# B&R Automation Studio project reAM250plc (part 4)

#### TcpPacketHandler.hpp
```cpp
/*++

Copyright (C) 2024 Institute for Machine Tools and Industrial Management
TUM School of Engineering and Design
Technical University of Munich

All rights reserved.

Redistribution and use in source and binary forms, with or without
modification, are permitted provided that the following conditions are met:
	* Redistributions of source code must retain the above copyright
	  notice, this list of conditions and the following disclaimer.
	* Redistributions in binary form must reproduce the above copyright
	  notice, this list of conditions and the following disclaimer in the
	  documentation and/or other materials provided with the distribution.
	* Neither the name of the Technical University of Munich nor the
	  names of its contributors may be used to endorse or promote products
	  derived from this software without specific prior written permission.

THIS SOFTWARE IS PROVIDED BY THE COPYRIGHT HOLDERS AND CONTRIBUTORS "AS IS" AND
ANY EXPRESS OR IMPLIED WARRANTIES, INCLUDING, BUT NOT LIMITED TO, THE IMPLIED
WARRANTIES OF MERCHANTABILITY AND FITNESS FOR A PARTICULAR PURPOSE ARE
DISCLAIMED. IN NO EVENT SHALL TECHNICAL UNIVERSITY OF MUNICH BE LIABLE FOR ANY
DIRECT, INDIRECT, INCIDENTAL, SPECIAL, EXEMPLARY, OR CONSEQUENTIAL DAMAGES
(INCLUDING, BUT NOT LIMITED TO, PROCUREMENT OF SUBSTITUTE GOODS OR SERVICES;
LOSS OF USE, DATA, OR PROFITS; OR BUSINESS INTERRUPTION) HOWEVER CAUSED AND
ON ANY THEORY OF LIABILITY, WHETHER IN CONTRACT, STRICT LIABILITY, OR TORT
(INCLUDING NEGLIGENCE OR OTHERWISE) ARISING IN ANY WAY OUT OF THE USE OF THIS
SOFTWARE, EVEN IF ADVISED OF THE POSSIBILITY OF SUCH DAMAGE.

*/

#ifndef __TCPPACKETHANDLER_HPP
#define __TCPPACKETHANDLER_HPP

#include "Framework.hpp"
#include <list>
#include <vector>
#include <map>
#include <array>
#define	TCP_MAX_PACKET_RESPONSESIZE (256 * 1024)

namespace BuRCPP {

	class CTcpPacketResponse {
		private:
			std::array<uint8_t, TCP_MAX_PACKET_RESPONSESIZE> m_Payload;

			uint32_t m_nSignature;
			uint32_t m_nClientID;
			uint32_t m_nSequenceID;
			uint32_t m_nCurrentSize;
			uint32_t m_nErrorCode;

		public:

			CTcpPacketResponse ();
			virtual ~CTcpPacketResponse ();

			void addUint8 (uint8_t nValue);
			void addUint16 (uint16_t nValue);
			void addUint32 (uint32_t nValue);
			void addInt8 (int8_t nValue);
			void addInt16 (int16_t nValue);
			void addInt32 (int32_t nValue);
			void addDouble (double nValue);
			void addString (const std::string & sValue);
			void addPayload (uint8_t * pData, uint32_t nDataSize);

			void setErrorCode (eErrorCode nErrorCode);

			void beginResponse (uint32_t nClientID, uint32_t nSequenceID, uint32_t nSignature);
			void clearPayload ();

			uint32_t getClientID ();
			uint32_t getSequenceID ();
			uint32_t getCurrentSize ();

			std::array<uint8_t, TCP_MAX_PACKET_RESPONSESIZE> & getPayload ();

			void buildHeader (TcpOutgoingMessageHeader & header);

	};

	class CTcpPacketHandler {
		private:

		public:

		CTcpPacketHandler ();
		virtual ~CTcpPacketHandler();

		virtual uint32_t getCommandID () = 0;

		virtual bool isBufferedCommand () = 0;

		virtual void handlePacket (TcpIncomingPayload * pPayload, CTcpPacketResponse * pResponse) = 0;

		static uint8_t readUint8FromPayload (TcpIncomingPayload * pPayload, uint32_t nOffset);
		static uint16_t readUint16FromPayload (TcpIncomingPayload * pPayload, uint32_t nOffset);
		static uint32_t readUint32FromPayload (TcpIncomingPayload * pPayload, uint32_t nOffset);

	};

	class CTcpPacketHandler_Direct : public CTcpPacketHandler {
		public:

			CTcpPacketHandler_Direct ();

			virtual ~CTcpPacketHandler_Direct();

			virtual bool isBufferedCommand () override;

	};

	class CTcpPacketRegistry {
		private:

		std::map<uint32_t, std::shared_ptr<CTcpPacketHandler>> m_Handlers;
		uint32_t m_nPacketSignature;
		bool m_bPerformChecksumCheck;

		public:

		CTcpPacketRegistry (uint32_t nPacketSignature);

		virtual ~CTcpPacketRegistry();

		void registerHandler (std::shared_ptr<CTcpPacketHandler> pPacketHandler);

		bool canHandlePacket (uint32_t nCommandID);

		bool handlePacket (uint8_t * pData, uint32_t nDataSize, CTcpPacketResponse * pResponse);

	};

}

#endif // __TCPPACKETHANDLER_HPP
```

#### TcpPacketHandler.cpp
```cpp
/*++

Copyright (C) 2024 Institute for Machine Tools and Industrial Management
TUM School of Engineering and Design
Technical University of Munich

All rights reserved.

Redistribution and use in source and binary forms, with or without
modification, are permitted provided that the following conditions are met:
	* Redistributions of source code must retain the above copyright
	  notice, this list of conditions and the following disclaimer.
	* Redistributions in binary form must reproduce the above copyright
	  notice, this list of conditions and the following disclaimer in the
	  documentation and/or other materials provided with the distribution.
	* Neither the name of the Technical University of Munich nor the
	  names of its contributors may be used to endorse or promote products
	  derived from this software without specific prior written permission.

THIS SOFTWARE IS PROVIDED BY THE COPYRIGHT HOLDERS AND CONTRIBUTORS "AS IS" AND
ANY EXPRESS OR IMPLIED WARRANTIES, INCLUDING, BUT NOT LIMITED TO, THE IMPLIED
WARRANTIES OF MERCHANTABILITY AND FITNESS FOR A PARTICULAR PURPOSE ARE
DISCLAIMED. IN NO EVENT SHALL TECHNICAL UNIVERSITY OF MUNICH BE LIABLE FOR ANY
DIRECT, INDIRECT, INCIDENTAL, SPECIAL, EXEMPLARY, OR CONSEQUENTIAL DAMAGES
(INCLUDING, BUT NOT LIMITED TO, PROCUREMENT OF SUBSTITUTE GOODS OR SERVICES;
LOSS OF USE, DATA, OR PROFITS; OR BUSINESS INTERRUPTION) HOWEVER CAUSED AND
ON ANY THEORY OF LIABILITY, WHETHER IN CONTRACT, STRICT LIABILITY, OR TORT
(INCLUDING NEGLIGENCE OR OTHERWISE) ARISING IN ANY WAY OUT OF THE USE OF THIS
SOFTWARE, EVEN IF ADVISED OF THE POSSIBILITY OF SUCH DAMAGE.

*/

#include "TcpPacketHandler.hpp"
#include "Utils.hpp"

#include <bur/plctypes.h>

#ifdef _DEFAULT_INCLUDES
#include <AsDefault.h>
#endif

#include <string.h>

namespace BuRCPP
{

	CTcpPacketResponse::CTcpPacketResponse ()
	:  m_nSignature (0), m_nClientID (0), m_nSequenceID (0), m_nCurrentSize (0), m_nErrorCode (0)
	{
	}

	CTcpPacketResponse::~CTcpPacketResponse ()
	{
	}

	void CTcpPacketResponse::addPayload (uint8_t * pData, uint32_t nDataSize)
	{
		if ((pData != nullptr) && (nDataSize > 0)) {
			if (nDataSize > TCP_MAX_PACKET_RESPONSESIZE)
				throw CException (eErrorCode::INVALIDPARAM, "invalid packet response payload size.");

			uint32_t nNewDataSize = m_nCurrentSize + nDataSize;
			if (nNewDataSize > TCP_MAX_PACKET_RESPONSESIZE)
				throw CException (eErrorCode::INVALIDPARAM, "packet response payload overflow.");

			uint8_t * pSource = pData;
			uint8_t * pTarget = &m_Payload.at (m_nCurrentSize);

			for (uint32_t nIndex = 0; nIndex < nDataSize; nIndex++)
			{
				*pTarget = *pSource;
				pTarget++;
				pSource++;
			}

			m_nCurrentSize += nDataSize;

		}
	}

	void CTcpPacketResponse::addUint8 (uint8_t nValue)
	{
		addPayload ((uint8_t*)&nValue, sizeof (nValue));
	}

	void CTcpPacketResponse::addUint16 (uint16_t nValue)
	{
		addPayload ((uint8_t*)&nValue, sizeof (nValue));
	}

	void CTcpPacketResponse::addUint32 (uint32_t nValue)
	{
		addPayload ((uint8_t*)&nValue, sizeof (nValue));
	}

	void CTcpPacketResponse::addInt8 (int8_t nValue)
	{
		addPayload ((uint8_t*)&nValue, sizeof (nValue));
	}

	void CTcpPacketResponse::addInt16 (int16_t nValue)
	{
		addPayload ((uint8_t*)&nValue, sizeof (nValue));
	}

	void CTcpPacketResponse::addInt32 (int32_t nValue)
	{
		addPayload ((uint8_t*)&nValue, sizeof (nValue));
	}

	void CTcpPacketResponse::addDouble (double nValue)
	{
		addPayload ((uint8_t*)&nValue, sizeof (nValue));
	}

	void CTcpPacketResponse::addString (const std::string & sValue)
	{
		uint32_t nLength = sValue.length ();
		addPayload ((uint8_t*) sValue.c_str (), nLength);
	}

	void CTcpPacketResponse::setErrorCode (eErrorCode nErrorCode)
	{
		m_nErrorCode = (uint32_t) nErrorCode;
	}

	void CTcpPacketResponse::beginResponse (uint32_t nClientID, uint32_t nSequenceID, uint32_t nSignature)
	{
		m_nClientID = nClientID;
		m_nSequenceID = nSequenceID;
		m_nCurrentSize = 0;
		m_nSignature = nSignature;
		m_nErrorCode = 0;
	}

	uint32_t CTcpPacketResponse::getClientID ()
	{
		return m_nClientID;
	}

	uint32_t CTcpPacketResponse::getSequenceID ()
	{
		return m_nSequenceID;
	}

	uint32_t CTcpPacketResponse::getCurrentSize ()
	{
		return m_nCurrentSize;
	}

	std::array<uint8_t, TCP_MAX_PACKET_RESPONSESIZE> & CTcpPacketResponse::getPayload ()
	{
		return m_Payload;
	}

	void CTcpPacketResponse::buildHeader (TcpOutgoingMessageHeader & header)
	{

		header.m_nClientId = m_nClientID;
		header.m_nPayloadLength = (uint32_t) m_nCurrentSize;
		header.m_nSequenceId = m_nSequenceID;
		header.m_nSignature = m_nSignature;
		header.m_nStatusCode = m_nErrorCode;

		if (m_nCurrentSize > 0) {
			header.m_nPayloadChecksum = CUtils::computeCRC32 (m_Payload.data (), (uint32_t) m_nCurrentSize);
		} else {
			header.m_nPayloadChecksum = 0;
		}
		header.m_nHeaderChecksum = CUtils::computeCRC32 ((uint8_t*) &header, sizeof (header) - 4);
	}

	void CTcpPacketResponse::clearPayload ()
	{
		m_nCurrentSize = 0;
	}

	CTcpPacketHandler::CTcpPacketHandler ()
	{
	}

	CTcpPacketHandler::~CTcpPacketHandler()
	{
	}

	uint8_t CTcpPacketHandler::readUint8FromPayload (TcpIncomingPayload * pPayload, uint32_t nOffset)
	{
		if (pPayload == nullptr)
			throw CException (eErrorCode::INVALIDPARAM, "invalid packet payload param.");
		if (nOffset >= sizeof (TcpIncomingPayload))
			throw CException (eErrorCode::INVALIDPAYLOADOFFSET, "invalid packet payload offset.");

		return pPayload->m_Data[nOffset];
	}

	uint16_t CTcpPacketHandler::readUint16FromPayload (TcpIncomingPayload * pPayload, uint32_t nOffset)
	{
		if (pPayload == nullptr)
			throw CException (eErrorCode::INVALIDPARAM, "invalid packet payload param.");
		if ((nOffset + sizeof (uint16_t)) > sizeof (TcpIncomingPayload))
			throw CException (eErrorCode::INVALIDPAYLOADOFFSET, "invalid packet payload offset.");

		return *((uint16_t*)&pPayload->m_Data[nOffset]);
	}

	uint32_t CTcpPacketHandler::readUint32FromPayload (TcpIncomingPayload * pPayload, uint32_t nOffset)
	{
		if (pPayload == nullptr)
			throw CException (eErrorCode::INVALIDPARAM, "invalid packet payload param.");
		if ((nOffset + sizeof (uint32_t)) > sizeof (TcpIncomingPayload))
			throw CException (eErrorCode::INVALIDPAYLOADOFFSET, "invalid packet payload offset.");

		return *((uint32_t*)&pPayload->m_Data[nOffset]);

	}

	CTcpPacketHandler_Direct::CTcpPacketHandler_Direct ()
	: CTcpPacketHandler ()
	{
	}

	CTcpPacketHandler_Direct::~CTcpPacketHandler_Direct()
	{
	}

	bool CTcpPacketHandler_Direct::isBufferedCommand ()
	{
		return false;
	}

	CTcpPacketRegistry::CTcpPacketRegistry (uint32_t nPacketSignature)
		: m_nPacketSignature (nPacketSignature), m_bPerformChecksumCheck(false)
	{
	}

	CTcpPacketRegistry::~CTcpPacketRegistry()
	{
	}

	void CTcpPacketRegistry::registerHandler (std::shared_ptr<CTcpPacketHandler> pPacketHandler)
	{
		if (pPacketHandler.get () == nullptr)
			throw CException (eErrorCode::INVALIDPARAM, "invalid packet handler param.");

		uint32_t nCommand = pPacketHandler->getCommandID ();
		if (canHandlePacket (nCommand))
			throw CException (eErrorCode::PACKETHANDLERALREADYREGISTERED, "packet handler already registered: " + std::to_string (nCommand));

		m_Handlers.insert (std::make_pair (nCommand, pPacketHandler));

	}

	bool CTcpPacketRegistry::canHandlePacket (uint32_t nCommandID)
	{
		auto iIter = m_Handlers.find (nCommandID);
		return (iIter != m_Handlers.end ());
	}

	bool CTcpPacketRegistry::handlePacket (uint8_t * pData, uint32_t nDataSize, CTcpPacketResponse * pResponse)
	{

		if (pData == nullptr)
			throw CException (eErrorCode::INVALIDPARAM, "invalid packet data param.");
		if (nDataSize != sizeof (TcpIncomingMessage))
			throw CException (eErrorCode::INVALIDPARAM, "invalid packet data size param.");
		if (pResponse == nullptr)
			throw CException (eErrorCode::INVALIDPARAM, "invalid packet response pointer.");

		TcpIncomingMessage * pMessage = (TcpIncomingMessage*) pData;
		uint32_t nCommandID = pMessage->m_nCommandId;

		if(pMessage->m_nSignature != m_nPacketSignature)
			return false;

		if (m_bPerformChecksumCheck) {

			uint32_t nChecksum = CUtils::computeCRC32 ((uint8_t*)pMessage, (uint32_t)sizeof(TcpIncomingMessage) - 4);
			if(pMessage->m_nChecksum != nChecksum)
				return false;
		}

		auto iIter = m_Handlers.find (nCommandID);
		if (iIter == m_Handlers.end ())
			return false;

		CTcpPacketHandler * pHandler = iIter->second.get();
		pResponse->beginResponse (pMessage->m_nClientId, pMessage->m_nSequenceId, pMessage->m_nSignature);
		try {
			pHandler->handlePacket (&pMessage->m_Payload, pResponse);
			return true;

		}
		catch (CException & E) {
			pResponse->setErrorCode (E.getCode ());
			pResponse->clearPayload ();
		}

	}

}
```

#### TcpListHandler.hpp
```cpp
/*++

Copyright (C) 2024 Institute for Machine Tools and Industrial Management
TUM School of Engineering and Design
Technical University of Munich

All rights reserved.

Redistribution and use in source and binary forms, with or without
modification, are permitted provided that the following conditions are met:
	* Redistributions of source code must retain the above copyright
	  notice, this list of conditions and the following disclaimer.
	* Redistributions in binary form must reproduce the above copyright
	  notice, this list of conditions and the following disclaimer in the
	  documentation and/or other materials provided with the distribution.
	* Neither the name of the Technical University of Munich nor the
	  names of its contributors may be used to endorse or promote products
	  derived from this software without specific prior written permission.

THIS SOFTWARE IS PROVIDED BY THE COPYRIGHT HOLDERS AND CONTRIBUTORS "AS IS" AND
ANY EXPRESS OR IMPLIED WARRANTIES, INCLUDING, BUT NOT LIMITED TO, THE IMPLIED
WARRANTIES OF MERCHANTABILITY AND FITNESS FOR A PARTICULAR PURPOSE ARE
DISCLAIMED. IN NO EVENT SHALL TECHNICAL UNIVERSITY OF MUNICH BE LIABLE FOR ANY
DIRECT, INDIRECT, INCIDENTAL, SPECIAL, EXEMPLARY, OR CONSEQUENTIAL DAMAGES
(INCLUDING, BUT NOT LIMITED TO, PROCUREMENT OF SUBSTITUTE GOODS OR SERVICES;
LOSS OF USE, DATA, OR PROFITS; OR BUSINESS INTERRUPTION) HOWEVER CAUSED AND
ON ANY THEORY OF LIABILITY, WHETHER IN CONTRACT, STRICT LIABILITY, OR TORT
(INCLUDING NEGLIGENCE OR OTHERWISE) ARISING IN ANY WAY OUT OF THE USE OF THIS
SOFTWARE, EVEN IF ADVISED OF THE POSSIBILITY OF SUCH DAMAGE.

*/

#ifndef __TCPSYSTEMSTATE_HPP
#define __TCPSYSTEMSTATE_HPP

#include "Framework.hpp"
#include "TcpPacketHandler.hpp"
#include "SignalHandler.hpp"

#include <memory>

#define LISTCONTEXT_SIGNALSLOTCOUNT 16

namespace BuRCPP {

	enum class eListEntryState : int32_t {
		InQueue = 0,
		InitialExecution = 1,
		CyclicExecution = 2,
		Finished = 3,
		ExecutionError = 4
	};

	enum class eListState : int32_t {
		ListInQueue = 0,
		ListInCreation = 1,
		ListFinished = 2,
		ExecutingList = 3,
		ExecutionFinished = 4,
		ExecutionError = 5
	};

	typedef struct _TcpListEntryContext {
		eListEntryState m_nEntryState;
		uint32_t m_nLifeTimeInMilliseconds;
		CSignalSendInstance * m_pSignalSlots[LISTCONTEXT_SIGNALSLOTCOUNT];
		uint8_t m_ContextData[32];
	} TcpListEntryContext;

	class CTcpListHandler;

	class CSignalHandlerRegistry {
		private:
		public:

			virtual CSignalHandler * findSignalHandler (const std::string & sStateMachineName, bool bMustExist) = 0;
	};

	class CPayloadEnvironment
	{
		private:

		TcpListEntryContext * m_pContext;
		TcpIncomingPayload * m_pPayload;
		CSignalHandlerRegistry * m_pSignalHandlerRegistry;

		public:

		CPayloadEnvironment (TcpListEntryContext * pContext, TcpIncomingPayload * pPayload, CSignalHandlerRegistry * pSignalHandlerRegistry);

		virtual ~CPayloadEnvironment ();

		eListEntryState getState ();

		bool isFirstCycle ();

		uint32_t getPayloadSize ();

		void readPayloadData (uint8_t * pTarget, uint32_t nAddress, uint32_t nByteCount);
		uint8_t readPayloadUint8 (uint32_t nAddress);
		uint16_t readPayloadUint16 (uint32_t nAddress);
		uint32_t readPayloadUint32 (uint32_t nAddress);
		int8_t readPayloadInt8 (uint32_t nAddress);
		int16_t readPayloadInt16 (uint32_t nAddress);
		int32_t readPayloadInt32 (uint32_t nAddress);
		double readPayloadDouble (uint32_t nAddress);
		float readPayloadFloat (uint32_t nAddress);

		uint32_t getContextSize ();

		void readContextData (uint8_t * pTarget, uint32_t nAddress, uint32_t nByteCount);
		uint8_t readContextUint8 (uint32_t nAddress);
		uint16_t readContextUint16 (uint32_t nAddress);
		uint32_t readContextUint32 (uint32_t nAddress);
		int8_t readContextInt8 (uint32_t nAddress);
		int16_t readContextInt16 (uint32_t nAddress);
		int32_t readContextInt32 (uint32_t nAddress);
		double readContextDouble (uint32_t nAddress);
		float readContextFloat (uint32_t nAddress);

		void writeContextData (uint8_t * pSource, uint32_t nAddress, uint32_t nByteCount);
		void writeContextUint8 (uint32_t nAddress, uint8_t nValue);
		void writeContextUint16 (uint32_t nAddress, uint16_t nValue);
		void writeContextUint32 (uint32_t nAddress, uint32_t nValue);
		void writeContextInt8 (uint32_t nAddress, int8_t nValue);
		void writeContextInt16 (uint32_t nAddress, int16_t nValue);
		void writeContextInt32 (uint32_t nAddress, int32_t nValue);
		void writeContextDouble (uint32_t nAddress, double dValue);
		void writeContextFloat (uint32_t nAddress, float dValue);

		void setLifetimeInMillseconds (uint32_t nLifeTimeInMilliseconds);

		CSignalSendInstance * prepareSignal (uint32_t nSignalSlotIndex, const std::string & sStateHandlerName, const std::string & sSignalName);
		CSignalSendInstance * getSignal (uint32_t nSignalSlotIndex, bool bMustExist);
		bool signalHasBeenProcessed (uint32_t nSignalSlotIndex);

	};

	class CTcpPacketHandler_Buffered : public CTcpPacketHandler {

		private:
		CTcpListHandler * m_pListHandler;

		public:

		CTcpPacketHandler_Buffered (CTcpListHandler * pListHandler);

		virtual ~CTcpPacketHandler_Buffered();

		virtual bool isBufferedCommand () override;

		virtual void handlePacket (TcpIncomingPayload * pPayload, CTcpPacketResponse * pResponse) override;

		virtual void enterExecution (CPayloadEnvironment * pEnvironment);

		virtual bool cyclicExecution (CPayloadEnvironment * pEnvironment);

	};

	struct _TcpListEntry;
	typedef struct _TcpListEntry TcpListEntry;

	struct _TcpList;
	typedef struct _TcpList TcpList;

	struct _TcpListEntry {
		CTcpPacketHandler_Buffered * m_PacketHandler;
		TcpIncomingPayload m_Payload;
		uint32_t m_nIndexInList;
		TcpListEntryContext m_ExecutionContext;
		TcpListEntry * m_pNext;
	};

	struct _TcpList {
		uint32_t m_nListId;
		uint32_t m_nEntryCount;
		eListState m_ListState;
		TcpListEntry * m_pFirstEntry;
		TcpListEntry * m_pLastEntry;
		TcpListEntry * m_pCurrentEntry;
		TcpList * m_pNextUnusedList;
	};

	class CTcpListHandler {

		private:
		std::vector<TcpListEntry> m_ListEntryBuffer;
		std::vector<TcpList> m_ListBuffer;
		TcpList * m_pUnusedLists;
		TcpListEntry * m_pUnusedListEntries;

		TcpList * m_pCurrentWriteList;

		TcpList * m_pCurrentExecutionList;

		CSignalHandlerRegistry * m_pSignalHandlerRegistry;

		void addEntryToList (TcpList *, CTcpPacketHandler_Buffered * pHandler, TcpIncomingPayload * pPayload);

		public:

		CTcpListHandler (uint32_t nListBufferSize, uint32_t nListEntryBufferSize, CSignalHandlerRegistry * pSignalHandlerRegistry);

		virtual ~CTcpListHandler ();

		void registerDefaultCommands (CTcpPacketRegistry * pPacketRegistry);

		uint32_t beginList ();
		TcpList * finishList ();
		TcpList* executeList (uint32_t nListID);
		TcpList* getListByID (uint32_t nListID, bool bListMustExist);

		bool hasCurrentList ();

		TcpListEntry * addCommandToCurrentList (CTcpPacketHandler_Buffered * pHandler, TcpIncomingPayload * pPayload);

		void handleCyclic ();

	};

}

#endif // __TCPSYSTEMSTATE_HPP
```

#### TcpListHandler.cpp
```cpp
/*++

Copyright (C) 2024 Institute for Machine Tools and Industrial Management
TUM School of Engineering and Design
Technical University of Munich

All rights reserved.

Redistribution and use in source and binary forms, with or without
modification, are permitted provided that the following conditions are met:
	* Redistributions of source code must retain the above copyright
	  notice, this list of conditions and the following disclaimer.
	* Redistributions in binary form must reproduce the above copyright
	  notice, this list of conditions and the following disclaimer in the
	  documentation and/or other materials provided with the distribution.
	* Neither the name of the Technical University of Munich nor the
	  names of its contributors may be used to endorse or promote products
	  derived from this software without specific prior written permission.

THIS SOFTWARE IS PROVIDED BY THE COPYRIGHT HOLDERS AND CONTRIBUTORS "AS IS" AND
ANY EXPRESS OR IMPLIED WARRANTIES, INCLUDING, BUT NOT LIMITED TO, THE IMPLIED
WARRANTIES OF MERCHANTABILITY AND FITNESS FOR A PARTICULAR PURPOSE ARE
DISCLAIMED. IN NO EVENT SHALL TECHNICAL UNIVERSITY OF MUNICH BE LIABLE FOR ANY
DIRECT, INDIRECT, INCIDENTAL, SPECIAL, EXEMPLARY, OR CONSEQUENTIAL DAMAGES
(INCLUDING, BUT NOT LIMITED TO, PROCUREMENT OF SUBSTITUTE GOODS OR SERVICES;
LOSS OF USE, DATA, OR PROFITS; OR BUSINESS INTERRUPTION) HOWEVER CAUSED AND
ON ANY THEORY OF LIABILITY, WHETHER IN CONTRACT, STRICT LIABILITY, OR TORT
(INCLUDING NEGLIGENCE OR OTHERWISE) ARISING IN ANY WAY OUT OF THE USE OF THIS
SOFTWARE, EVEN IF ADVISED OF THE POSSIBILITY OF SUCH DAMAGE.

*/

#include "TcpListHandler.hpp"

#include <cstring>

namespace BuRCPP {

	CPayloadEnvironment::CPayloadEnvironment (TcpListEntryContext * pContext, TcpIncomingPayload * pPayload, CSignalHandlerRegistry * pSignalHandlerRegistry)
		: m_pContext (pContext), m_pPayload (pPayload), m_pSignalHandlerRegistry (pSignalHandlerRegistry)
	{
		if ((pContext == nullptr) || (pPayload == nullptr) || (pSignalHandlerRegistry == nullptr))
			throw CException (eErrorCode::INVALIDPARAM, "invalid payload environment parameters");

	}

	CPayloadEnvironment::~CPayloadEnvironment ()
	{
	}

	eListEntryState CPayloadEnvironment::getState ()
	{
		return m_pContext->m_nEntryState;
	}

	bool CPayloadEnvironment::isFirstCycle ()
	{
		return m_pContext->m_nEntryState == eListEntryState::InitialExecution;
	}

	uint32_t CPayloadEnvironment::getPayloadSize ()
	{
		return sizeof (TcpIncomingPayload);
	}

	void CPayloadEnvironment::readPayloadData (uint8_t * pTarget, uint32_t nAddress, uint32_t nByteCount)
	{
		if (nByteCount == 0)
			return;

		if (pTarget == nullptr)
			throw CException (eErrorCode::INVALIDPARAM, "invalid read payload target parameter");

		if (nAddress >=  sizeof (TcpIncomingPayload))
			throw CException (eErrorCode::INVALIDPAYLOADADDRESS, "invalid payload address");

		if (nByteCount >=  sizeof (TcpIncomingPayload))
			throw CException (eErrorCode::INVALIDPAYLOADREADOPERATION, "invalid payload read size");
		if ((nAddress + nByteCount) > sizeof (TcpIncomingPayload))
			throw CException (eErrorCode::INVALIDPAYLOADREADOPERATION, "payload read buffer overflow");

		for (uint32_t nIndex = 0; nIndex < nByteCount; nIndex++)
			pTarget[nIndex] = m_pPayload->m_Data[nAddress + nIndex];

	}

	uint8_t CPayloadEnvironment::readPayloadUint8 (uint32_t nAddress)
	{
		uint8_t nResult = 0;
		readPayloadData ((uint8_t*)&nResult, nAddress, sizeof (nResult));
		return nResult;
	}

	uint16_t CPayloadEnvironment::readPayloadUint16 (uint32_t nAddress)
	{
		uint16_t nResult = 0;
		readPayloadData ((uint8_t*)&nResult, nAddress, sizeof (nResult));
		return nResult;
	}

	uint32_t CPayloadEnvironment::readPayloadUint32 (uint32_t nAddress)
	{
		uint32_t nResult = 0;
		readPayloadData ((uint8_t*)&nResult, nAddress, sizeof (nResult));
		return nResult;
	}

	int8_t CPayloadEnvironment::readPayloadInt8 (uint32_t nAddress)
	{
		int8_t nResult = 0;
		readPayloadData ((uint8_t*)&nResult, nAddress, sizeof (nResult));
		return nResult;
	}

	int16_t CPayloadEnvironment::readPayloadInt16 (uint32_t nAddress)
	{
		int16_t nResult = 0;
		readPayloadData ((uint8_t*)&nResult, nAddress, sizeof (nResult));
		return nResult;
	}

	int32_t CPayloadEnvironment::readPayloadInt32 (uint32_t nAddress)
	{
		uint32_t nResult = 0;
		readPayloadData ((uint8_t*)&nResult, nAddress, sizeof (nResult));
		return nResult;

	}

	double CPayloadEnvironment::readPayloadDouble (uint32_t nAddress)
	{
		double dResult = 0.0;
		readPayloadData ((uint8_t*)&dResult, nAddress, sizeof (dResult));
		return dResult;

	}

	float CPayloadEnvironment::readPayloadFloat (uint32_t nAddress)
	{
		float fResult = 0.0;
		readPayloadData ((uint8_t*)&fResult, nAddress, sizeof (fResult));
		return fResult;

	}

	uint32_t CPayloadEnvironment::getContextSize ()
	{
		return sizeof (m_pContext->m_ContextData);
	}

	void CPayloadEnvironment::readContextData (uint8_t * pTarget, uint32_t nAddress, uint32_t nByteCount)
	{
	}

	uint8_t CPayloadEnvironment::readContextUint8 (uint32_t nAddress)
	{

	}

	uint16_t CPayloadEnvironment::readContextUint16 (uint32_t nAddress)
	{

	}

	uint32_t CPayloadEnvironment::readContextUint32 (uint32_t nAddress)
	{

	}

	int8_t CPayloadEnvironment::readContextInt8 (uint32_t nAddress)
	{

	}

	int16_t CPayloadEnvironment::readContextInt16 (uint32_t nAddress)
	{

	}

	int32_t CPayloadEnvironment::readContextInt32 (uint32_t nAddress)
	{

	}

	double CPayloadEnvironment::readContextDouble (uint32_t nAddress)
	{

	}

	float CPayloadEnvironment::readContextFloat (uint32_t nAddress)
	{

	}

	void CPayloadEnvironment::writeContextData (uint8_t * pSource, uint32_t nAddress, uint32_t nByteCount)
	{

	}

	void CPayloadEnvironment::writeContextUint8 (uint32_t nAddress, uint8_t nValue)
	{
	}

	void CPayloadEnvironment::writeContextUint16 (uint32_t nAddress, uint16_t nValue)
	{
	}

	void CPayloadEnvironment::writeContextUint32 (uint32_t nAddress, uint32_t nValue)
	{
	}

	void CPayloadEnvironment::writeContextInt8 (uint32_t nAddress, int8_t nValue)
	{
	}

	void CPayloadEnvironment::writeContextInt16 (uint32_t nAddress, int16_t nValue)
	{
	}

	void CPayloadEnvironment::writeContextInt32 (uint32_t nAddress, int32_t nValue)
	{
	}

	void CPayloadEnvironment::writeContextDouble (uint32_t nAddress, double dValue)
	{
	}

	void CPayloadEnvironment::writeContextFloat (uint32_t nAddress, float dValue)
	{
	}

	void CPayloadEnvironment::setLifetimeInMillseconds (uint32_t nLifeTimeInMilliseconds)
	{
		m_pContext->m_nLifeTimeInMilliseconds = nLifeTimeInMilliseconds;
	}

	CSignalSendInstance * CPayloadEnvironment::prepareSignal (uint32_t nSignalSlotIndex, const std::string & sStateHandlerName, const std::string & sSignalName)
	{
		if (nSignalSlotIndex >= LISTCONTEXT_SIGNALSLOTCOUNT)
			throw CException (eErrorCode::INVALIDSIGNALSLOTINDEX, "invalid payload signal slot index: " + std::to_string (nSignalSlotIndex));

		if (m_pContext->m_pSignalSlots[nSignalSlotIndex] != nullptr)
			throw CException (eErrorCode::PAYLOADSIGNALSLOTALREADYTAKEN, "signal slot already taken: " + std::to_string (nSignalSlotIndex));

		auto pSignalHandler = m_pSignalHandlerRegistry->findSignalHandler (sStateHandlerName, true);

		CSignalSendInstance * pSignalInstance = pSignalHandler->prepareSignal (sSignalName);

		m_pContext->m_pSignalSlots[nSignalSlotIndex] = pSignalInstance;

		return pSignalInstance;
	}

	CSignalSendInstance * CPayloadEnvironment::getSignal (uint32_t nSignalSlotIndex, bool bMustExist)
	{
		if (nSignalSlotIndex >= LISTCONTEXT_SIGNALSLOTCOUNT)
			throw CException (eErrorCode::INVALIDSIGNALSLOTINDEX, "invalid payload signal slot index: " + std::to_string (nSignalSlotIndex));

		CSignalSendInstance * pSignalInstance =	m_pContext->m_pSignalSlots[nSignalSlotIndex];
		if ((pSignalInstance == nullptr) && bMustExist)
			throw CException (eErrorCode::SIGNALSLOTISEMPTY, "payload signal slot is empty: " + std::to_string (nSignalSlotIndex));

		return pSignalInstance;
	}

	bool CPayloadEnvironment::signalHasBeenProcessed (uint32_t nSignalSlot)
	{
		CSignalSendInstance * pSignalInstance = getSignal (nSignalSlot, true);
		return pSignalInstance->signalHasBeenProcessed ();
	}

	class CTcpPacketHandler_BeginList : public CTcpPacketHandler_Direct {
		private:
			CTcpListHandler* m_pListHandler;

		public:

			CTcpPacketHandler_BeginList (CTcpListHandler * pListHandler)
			: CTcpPacketHandler_Direct (), m_pListHandler (pListHandler)
				{
				}

			virtual ~CTcpPacketHandler_BeginList ()
			{
			}

			virtual uint32_t getCommandID () override
			{
				return COMMAND_DEFAULT_BEGINLIST;
			}

			void handlePacket (TcpIncomingPayload * pPayload, CTcpPacketResponse * pResponse) override
			{
				beginListCalled++;
				pResponse->addUint32(m_pListHandler->beginList ());
			}

	};

	class CTcpPacketHandler_FinishList : public CTcpPacketHandler_Direct {
		private:
		CTcpListHandler* m_pListHandler;

		public:

		CTcpPacketHandler_FinishList (CTcpListHandler * pListHandler)
			: CTcpPacketHandler_Direct (), m_pListHandler (pListHandler)
		{
		}

		virtual ~CTcpPacketHandler_FinishList ()
		{
		}

		virtual uint32_t getCommandID () override
		{
			return COMMAND_DEFAULT_FINISHLIST;
		}

			void handlePacket (TcpIncomingPayload * pPayload, CTcpPacketResponse * pResponse) override
			{
				finishListCalled++;
				TcpList* pList = m_pListHandler->finishList ();
				pResponse->addUint32(pList->m_nListId);
				pResponse->addUint32(pList->m_nEntryCount);
			}

	};

	class CTcpPacketHandler_ExecuteList : public CTcpPacketHandler_Direct {
		private:
		CTcpListHandler* m_pListHandler;

		public:

		CTcpPacketHandler_ExecuteList (CTcpListHandler * pListHandler)
			: CTcpPacketHandler_Direct (), m_pListHandler (pListHandler)
		{
		}

		virtual ~CTcpPacketHandler_ExecuteList ()
		{
		}

		virtual uint32_t getCommandID () override
		{
			return COMMAND_DEFAULT_EXECUTELIST;
		}

		void handlePacket (TcpIncomingPayload * pPayload, CTcpPacketResponse * pResponse) override
		{
			uint32_t nListID = readUint32FromPayload (pPayload, 0);
			TcpList * pList = m_pListHandler->executeList (nListID);

			pResponse->addUint32(pList->m_nEntryCount);
		}
	};

		class CTcpPacketHandler_ListStatus : public CTcpPacketHandler_Direct {
			private:
			CTcpListHandler* m_pListHandler;

			public:

				CTcpPacketHandler_ListStatus (CTcpListHandler * pListHandler)
					: CTcpPacketHandler_Direct (), m_pListHandler (pListHandler)
				{
				}

				virtual ~CTcpPacketHandler_ListStatus ()
				{
				}

				virtual uint32_t getCommandID () override
				{
					return COMMAND_DEFAULT_LISTSTATUS;
				}

				void handlePacket (TcpIncomingPayload * pPayload, CTcpPacketResponse * pResponse) override
				{
					uint32_t nListID = readUint32FromPayload (pPayload, 0);
					TcpList * pList = m_pListHandler->getListByID (nListID, false);

					if (pList != nullptr) {
						pResponse->addUint32(pList->m_nListId);
						pResponse->addUint32((uint32_t)pList->m_ListState);
						pResponse->addUint32(pList->m_nEntryCount);
						if (pList->m_pCurrentEntry != nullptr) {
							pResponse->addUint32(pList->m_pCurrentEntry->m_nIndexInList);
						} else {
							pResponse->addUint32(0);
						}

					} else {
						pResponse->addUint32(0);
						pResponse->addUint32(0);
						pResponse->addUint32(0);
						pResponse->addUint32(0);
					}

				}

	};

CTcpPacketHandler_Buffered::CTcpPacketHandler_Buffered (CTcpListHandler * pListHandler)
	: CTcpPacketHandler (), m_pListHandler (pListHandler)
{
}

CTcpPacketHandler_Buffered::~CTcpPacketHandler_Buffered()
{
}

bool CTcpPacketHandler_Buffered::isBufferedCommand ()
{
	return true;
}

void CTcpPacketHandler_Buffered::handlePacket (TcpIncomingPayload * pPayload, CTcpPacketResponse * pResponse)
{
	TcpListEntry* pNewEntry = m_pListHandler->addCommandToCurrentList (this, pPayload);
	pResponse->addUint32(pNewEntry->m_nIndexInList);

}

void CTcpPacketHandler_Buffered::enterExecution (CPayloadEnvironment * pEnvironment)
{

}

bool CTcpPacketHandler_Buffered::cyclicExecution (CPayloadEnvironment * pEnvironment)
{
	return true;
}

	CTcpListHandler::CTcpListHandler (uint32_t nListBufferSize, uint32_t nListEntryBufferSize, CSignalHandlerRegistry * pSignalHandlerRegistry)
	: m_pUnusedLists (nullptr), m_pUnusedListEntries (nullptr), m_pCurrentWriteList (nullptr), m_pCurrentExecutionList (nullptr), m_pSignalHandlerRegistry (pSignalHandlerRegistry)
	{

		if (pSignalHandlerRegistry == nullptr)
			throw std::runtime_error ("invalid signal handler registry param");

		m_ListEntryBuffer.resize (nListEntryBufferSize);
		m_ListBuffer.resize (nListBufferSize);

		uint32_t nListIndex = nListBufferSize;
		while (nListIndex > 0) {
			nListIndex--;

			auto pList = &m_ListBuffer[nListIndex];
			pList->m_nListId = nListIndex + 1;
			pList->m_nEntryCount = 0;
			pList->m_pLastEntry = nullptr;
			pList->m_pFirstEntry = nullptr;
			pList->m_pCurrentEntry = nullptr;
			pList->m_ListState = eListState::ListInQueue;

			pList->m_pNextUnusedList = m_pUnusedLists;
			m_pUnusedLists = pList;

		}

		uint32_t nListEntryIndex = nListEntryBufferSize;
		while (nListEntryIndex > 0) {
			nListEntryIndex--;

			auto pListEntry = &m_ListEntryBuffer[nListEntryIndex];
			pListEntry->m_pNext = m_pUnusedListEntries;
			pListEntry->m_PacketHandler = nullptr;
			pListEntry->m_nIndexInList = 0;
			memset ((void*) &pListEntry->m_Payload, 0, sizeof (pListEntry->m_Payload));
			m_pUnusedListEntries = pListEntry;

		}
	}

	CTcpListHandler::~CTcpListHandler ()
	{
	}

	void CTcpListHandler::registerDefaultCommands (CTcpPacketRegistry * pPacketRegistry)
	{
		if (pPacketRegistry == nullptr)
			throw CException (eErrorCode::INVALIDPARAM, "invalid packet registry parameter");

		pPacketRegistry->registerHandler (std::make_shared<CTcpPacketHandler_BeginList> (this));
		pPacketRegistry->registerHandler (std::make_shared<CTcpPacketHandler_FinishList> (this));
		pPacketRegistry->registerHandler (std::make_shared<CTcpPacketHandler_ExecuteList> (this));
		pPacketRegistry->registerHandler (std::make_shared<CTcpPacketHandler_ListStatus> (this));

	}

	uint32_t CTcpListHandler::beginList ()
	{
		if (m_pUnusedLists == nullptr)
			throw CException (eErrorCode::TOOMANYOPENLISTS, "too many open lists!");

		if (m_pUnusedLists->m_ListState != eListState::ListInQueue)
			throw CException (eErrorCode::LISTISNOTINQUEUE, "list is not in queue!");

		m_pCurrentWriteList = m_pUnusedLists;
		m_pUnusedLists = m_pUnusedLists->m_pNextUnusedList;

		m_pCurrentWriteList->m_nEntryCount = 0;
		m_pCurrentWriteList->m_pCurrentEntry = nullptr;
		m_pCurrentWriteList->m_pFirstEntry = nullptr;
		m_pCurrentWriteList->m_pLastEntry = nullptr;
		m_pCurrentWriteList->m_pNextUnusedList = nullptr;
		m_pCurrentWriteList->m_ListState = eListState::ListInCreation;

		return m_pCurrentWriteList->m_nListId;
	}

	TcpList* CTcpListHandler::finishList ()
	{

		if (m_pCurrentWriteList == nullptr)
			throw CException (eErrorCode::NOTWRITINGTOANYLIST, "not writing to any list!");
		if (m_pCurrentWriteList->m_ListState != eListState::ListInCreation)
			throw CException (eErrorCode::NOTINLISTCREATION, "list not in creation!");
		if (m_pCurrentWriteList->m_pFirstEntry == nullptr)
			throw CException (eErrorCode::LISTISEMPTY, "list is empty!");

		auto pList = m_pCurrentWriteList;
		m_pCurrentWriteList = nullptr;

		pList->m_ListState = eListState::ListFinished;
		return pList;
	}

	TcpList* CTcpListHandler::getListByID (uint32_t nListID, bool bListMustExist)
	{
		TcpList * pList = nullptr;
		if ((nListID > 0) || (nListID <= m_ListBuffer.size ())) {
			pList = &m_ListBuffer.at (nListID - 1);
			if (pList->m_ListState == eListState::ListInQueue)
				pList = nullptr;
		}

		if ((pList == nullptr) && bListMustExist)
			throw CException (eErrorCode::LISTDOESNOTEXIST, "list does not exist");

		return pList;
	}

	TcpList* CTcpListHandler::executeList (uint32_t nListID)
	{
		m_pCurrentExecutionList = nullptr;

		if ((nListID == 0) || (nListID > m_ListBuffer.size ()))
			throw CException (eErrorCode::INVALIDLISTID, "invalid list ID");

		auto pList = &m_ListBuffer.at (nListID - 1);
		if (pList->m_ListState != eListState::ListFinished)
			throw CException (eErrorCode::LISTISNOTFINISHED, "list is not in finished!");
		if (pList->m_pFirstEntry == nullptr)
			throw CException (eErrorCode::LISTISEMPTY, "list is empty!");

		m_pCurrentExecutionList = pList;
		m_pCurrentExecutionList->m_pCurrentEntry = m_pCurrentExecutionList->m_pFirstEntry;
		m_pCurrentExecutionList->m_ListState = eListState::ExecutingList;

		return m_pCurrentExecutionList;
	}

	bool CTcpListHandler::hasCurrentList ()
	{
		return (m_pCurrentWriteList != nullptr);
	}

	TcpListEntry* CTcpListHandler::addCommandToCurrentList (CTcpPacketHandler_Buffered * pHandler, TcpIncomingPayload * pPayload)
	{
		if (pHandler == nullptr)
			throw CException (eErrorCode::INVALIDPARAM, "invalid packet handler parameter");
		if (pPayload == nullptr)
			throw CException (eErrorCode::INVALIDPAYLOAD, "invalid payload.");
		if (m_pCurrentWriteList == nullptr)
			throw CException (eErrorCode::NOLISTTOWRITETO, "no list to write to.");
		if (m_pUnusedListEntries == nullptr)
			throw CException (eErrorCode::NOLISTENTRIESLEFT, "no list entries left");

		auto pNewListEntry = m_pUnusedListEntries;
		m_pUnusedListEntries = m_pUnusedListEntries->m_pNext;

		pNewListEntry->m_PacketHandler = pHandler;
		pNewListEntry->m_Payload = *pPayload;
		pNewListEntry->m_pNext = nullptr;
		pNewListEntry->m_nIndexInList = m_pCurrentWriteList->m_nEntryCount;

		memset ((void*)&pNewListEntry->m_ExecutionContext, 0, sizeof (pNewListEntry->m_ExecutionContext));
		pNewListEntry->m_ExecutionContext.m_nEntryState = eListEntryState::InQueue;

		m_pCurrentWriteList->m_nEntryCount++;
		if (m_pCurrentWriteList->m_pFirstEntry == nullptr)
			m_pCurrentWriteList->m_pFirstEntry = pNewListEntry;
		if (m_pCurrentWriteList->m_pLastEntry != nullptr)
			m_pCurrentWriteList->m_pLastEntry->m_pNext = pNewListEntry;
		m_pCurrentWriteList->m_pLastEntry = pNewListEntry;

		bufferedListEntries++;

		return pNewListEntry;
	}

	void CTcpListHandler::handleCyclic ()
	{
		if (m_pCurrentExecutionList != nullptr) {

			auto pEntryToExecute = m_pCurrentExecutionList->m_pCurrentEntry;
			if (pEntryToExecute != nullptr) {
				switch (pEntryToExecute->m_ExecutionContext.m_nEntryState) {
					case eListEntryState::InQueue:
					{
						pEntryToExecute->m_ExecutionContext.m_nEntryState = eListEntryState::InitialExecution;
						break;
					}

					case eListEntryState::InitialExecution:
					{
						try {

							if (pEntryToExecute->m_PacketHandler == nullptr)
								throw CException (eErrorCode::INTERNALLISTERROR, "internal list error");

							CPayloadEnvironment environment (&pEntryToExecute->m_ExecutionContext, &pEntryToExecute->m_Payload, m_pSignalHandlerRegistry);

							pEntryToExecute->m_PacketHandler->enterExecution (&environment);
							pEntryToExecute->m_ExecutionContext.m_nEntryState = eListEntryState::CyclicExecution;

						} catch (...) {
							pEntryToExecute->m_ExecutionContext.m_nEntryState = eListEntryState::ExecutionError;
						}

						break;
					}

					case eListEntryState::CyclicExecution:
					{
						try {

							if (pEntryToExecute->m_PacketHandler == nullptr)
								throw CException (eErrorCode::INTERNALLISTERROR, "internal list error");

							CPayloadEnvironment environment (&pEntryToExecute->m_ExecutionContext, &pEntryToExecute->m_Payload, m_pSignalHandlerRegistry);

							bool bIsFinished = pEntryToExecute->m_PacketHandler->cyclicExecution (&environment);
							if (bIsFinished) {
								pEntryToExecute->m_ExecutionContext.m_nEntryState = eListEntryState::Finished;
							} else {
								pEntryToExecute->m_ExecutionContext.m_nEntryState = eListEntryState::CyclicExecution;
							}

						} catch (...) {
							pEntryToExecute->m_ExecutionContext.m_nEntryState = eListEntryState::ExecutionError;
						}

						break;
					}

					case eListEntryState::Finished:
					{
						m_pCurrentExecutionList->m_pCurrentEntry = pEntryToExecute->m_pNext;
						break;
					}

					case eListEntryState::ExecutionError:
					{
						m_pCurrentExecutionList = nullptr;
						break;
					}

				}

			}

		}
	}

}
```

#### Utils.hpp
```cpp
/*++

Copyright (C) 2024 Institute for Machine Tools and Industrial Management
TUM School of Engineering and Design
Technical University of Munich

All rights reserved.

Redistribution and use in source and binary forms, with or without
modification, are permitted provided that the following conditions are met:
	* Redistributions of source code must retain the above copyright
	  notice, this list of conditions and the following disclaimer.
	* Redistributions in binary form must reproduce the above copyright
	  notice, this list of conditions and the following disclaimer in the
	  documentation and/or other materials provided with the distribution.
	* Neither the name of the Technical University of Munich nor the
	  names of its contributors may be used to endorse or promote products
	  derived from this software without specific prior written permission.

THIS SOFTWARE IS PROVIDED BY THE COPYRIGHT HOLDERS AND CONTRIBUTORS "AS IS" AND
ANY EXPRESS OR IMPLIED WARRANTIES, INCLUDING, BUT NOT LIMITED TO, THE IMPLIED
WARRANTIES OF MERCHANTABILITY AND FITNESS FOR A PARTICULAR PURPOSE ARE
DISCLAIMED. IN NO EVENT SHALL TECHNICAL UNIVERSITY OF MUNICH BE LIABLE FOR ANY
DIRECT, INDIRECT, INCIDENTAL, SPECIAL, EXEMPLARY, OR CONSEQUENTIAL DAMAGES
(INCLUDING, BUT NOT LIMITED TO, PROCUREMENT OF SUBSTITUTE GOODS OR SERVICES;
LOSS OF USE, DATA, OR PROFITS; OR BUSINESS INTERRUPTION) HOWEVER CAUSED AND
ON ANY THEORY OF LIABILITY, WHETHER IN CONTRACT, STRICT LIABILITY, OR TORT
(INCLUDING NEGLIGENCE OR OTHERWISE) ARISING IN ANY WAY OUT OF THE USE OF THIS
SOFTWARE, EVEN IF ADVISED OF THE POSSIBILITY OF SUCH DAMAGE.

*/

#ifndef __UTILS_HPP
#define __UTILS_HPP

#include "Framework.hpp"
#include <memory>

namespace BuRCPP {

	class CUtils {

	public:

		static uint32_t computeCRC32 (uint8_t * pBuf, uint32_t len);

		static void writeStringVariable(const std::string & sString, char * pVariable, uint32_t nCount);

	};

}

#endif // __UTILS_HPP
```

#### Utils.cpp
```cpp
/*++

Copyright (C) 2024 Institute for Machine Tools and Industrial Management
TUM School of Engineering and Design
Technical University of Munich

All rights reserved.

Redistribution and use in source and binary forms, with or without
modification, are permitted provided that the following conditions are met:
	* Redistributions of source code must retain the above copyright
	  notice, this list of conditions and the following disclaimer.
	* Redistributions in binary form must reproduce the above copyright
	  notice, this list of conditions and the following disclaimer in the
	  documentation and/or other materials provided with the distribution.
	* Neither the name of the Technical University of Munich nor the
	  names of its contributors may be used to endorse or promote products
	  derived from this software without specific prior written permission.

THIS SOFTWARE IS PROVIDED BY THE COPYRIGHT HOLDERS AND CONTRIBUTORS "AS IS" AND
ANY EXPRESS OR IMPLIED WARRANTIES, INCLUDING, BUT NOT LIMITED TO, THE IMPLIED
WARRANTIES OF MERCHANTABILITY AND FITNESS FOR A PARTICULAR PURPOSE ARE
DISCLAIMED. IN NO EVENT SHALL TECHNICAL UNIVERSITY OF MUNICH BE LIABLE FOR ANY
DIRECT, INDIRECT, INCIDENTAL, SPECIAL, EXEMPLARY, OR CONSEQUENTIAL DAMAGES
(INCLUDING, BUT NOT LIMITED TO, PROCUREMENT OF SUBSTITUTE GOODS OR SERVICES;
LOSS OF USE, DATA, OR PROFITS; OR BUSINESS INTERRUPTION) HOWEVER CAUSED AND
ON ANY THEORY OF LIABILITY, WHETHER IN CONTRACT, STRICT LIABILITY, OR TORT
(INCLUDING NEGLIGENCE OR OTHERWISE) ARISING IN ANY WAY OUT OF THE USE OF THIS
SOFTWARE, EVEN IF ADVISED OF THE POSSIBILITY OF SUCH DAMAGE.

*/

#include "Utils.hpp"

namespace BuRCPP {

	const uint32_t crc_table[256] = {
		0x00000000L, 0x77073096L, 0xee0e612cL, 0x990951baL, 0x076dc419L,
		0x706af48fL, 0xe963a535L, 0x9e6495a3L, 0x0edb8832L, 0x79dcb8a4L,
		0xe0d5e91eL, 0x97d2d988L, 0x09b64c2bL, 0x7eb17cbdL, 0xe7b82d07L,
		0x90bf1d91L, 0x1db71064L, 0x6ab020f2L, 0xf3b97148L, 0x84be41deL,
		0x1adad47dL, 0x6ddde4ebL, 0xf4d4b551L, 0x83d385c7L, 0x136c9856L,
		0x646ba8c0L, 0xfd62f97aL, 0x8a65c9ecL, 0x14015c4fL, 0x63066cd9L,
		0xfa0f3d63L, 0x8d080df5L, 0x3b6e20c8L, 0x4c69105eL, 0xd56041e4L,
		0xa2677172L, 0x3c03e4d1L, 0x4b04d447L, 0xd20d85fdL, 0xa50ab56bL,
		0x35b5a8faL, 0x42b2986cL, 0xdbbbc9d6L, 0xacbcf940L, 0x32d86ce3L,
		0x45df5c75L, 0xdcd60dcfL, 0xabd13d59L, 0x26d930acL, 0x51de003aL,
		0xc8d75180L, 0xbfd06116L, 0x21b4f4b5L, 0x56b3c423L, 0xcfba9599L,
		0xb8bda50fL, 0x2802b89eL, 0x5f058808L, 0xc60cd9b2L, 0xb10be924L,
		0x2f6f7c87L, 0x58684c11L, 0xc1611dabL, 0xb6662d3dL, 0x76dc4190L,
		0x01db7106L, 0x98d220bcL, 0xefd5102aL, 0x71b18589L, 0x06b6b51fL,
		0x9fbfe4a5L, 0xe8b8d433L, 0x7807c9a2L, 0x0f00f934L, 0x9609a88eL,
		0xe10e9818L, 0x7f6a0dbbL, 0x086d3d2dL, 0x91646c97L, 0xe6635c01L,
		0x6b6b51f4L, 0x1c6c6162L, 0x856530d8L, 0xf262004eL, 0x6c0695edL,
		0x1b01a57bL, 0x8208f4c1L, 0xf50fc457L, 0x65b0d9c6L, 0x12b7e950L,
		0x8bbeb8eaL, 0xfcb9887cL, 0x62dd1ddfL, 0x15da2d49L, 0x8cd37cf3L,
		0xfbd44c65L, 0x4db26158L, 0x3ab551ceL, 0xa3bc0074L, 0xd4bb30e2L,
		0x4adfa541L, 0x3dd895d7L, 0xa4d1c46dL, 0xd3d6f4fbL, 0x4369e96aL,
		0x346ed9fcL, 0xad678846L, 0xda60b8d0L, 0x44042d73L, 0x33031de5L,
		0xaa0a4c5fL, 0xdd0d7cc9L, 0x5005713cL, 0x270241aaL, 0xbe0b1010L,
		0xc90c2086L, 0x5768b525L, 0x206f85b3L, 0xb966d409L, 0xce61e49fL,
		0x5edef90eL, 0x29d9c998L, 0xb0d09822L, 0xc7d7a8b4L, 0x59b33d17L,
		0x2eb40d81L, 0xb7bd5c3bL, 0xc0ba6cadL, 0xedb88320L, 0x9abfb3b6L,
		0x03b6e20cL, 0x74b1d29aL, 0xead54739L, 0x9dd277afL, 0x04db2615L,
		0x73dc1683L, 0xe3630b12L, 0x94643b84L, 0x0d6d6a3eL, 0x7a6a5aa8L,
		0xe40ecf0bL, 0x9309ff9dL, 0x0a00ae27L, 0x7d079eb1L, 0xf00f9344L,
		0x8708a3d2L, 0x1e01f268L, 0x6906c2feL, 0xf762575dL, 0x806567cbL,
		0x196c3671L, 0x6e6b06e7L, 0xfed41b76L, 0x89d32be0L, 0x10da7a5aL,
		0x67dd4accL, 0xf9b9df6fL, 0x8ebeeff9L, 0x17b7be43L, 0x60b08ed5L,
		0xd6d6a3e8L, 0xa1d1937eL, 0x38d8c2c4L, 0x4fdff252L, 0xd1bb67f1L,
		0xa6bc5767L, 0x3fb506ddL, 0x48b2364bL, 0xd80d2bdaL, 0xaf0a1b4cL,
		0x36034af6L, 0x41047a60L, 0xdf60efc3L, 0xa867df55L, 0x316e8eefL,
		0x4669be79L, 0xcb61b38cL, 0xbc66831aL, 0x256fd2a0L, 0x5268e236L,
		0xcc0c7795L, 0xbb0b4703L, 0x220216b9L, 0x5505262fL, 0xc5ba3bbeL,
		0xb2bd0b28L, 0x2bb45a92L, 0x5cb36a04L, 0xc2d7ffa7L, 0xb5d0cf31L,
		0x2cd99e8bL, 0x5bdeae1dL, 0x9b64c2b0L, 0xec63f226L, 0x756aa39cL,
		0x026d930aL, 0x9c0906a9L, 0xeb0e363fL, 0x72076785L, 0x05005713L,
		0x95bf4a82L, 0xe2b87a14L, 0x7bb12baeL, 0x0cb61b38L, 0x92d28e9bL,
		0xe5d5be0dL, 0x7cdcefb7L, 0x0bdbdf21L, 0x86d3d2d4L, 0xf1d4e242L,
		0x68ddb3f8L, 0x1fda836eL, 0x81be16cdL, 0xf6b9265bL, 0x6fb077e1L,
		0x18b74777L, 0x88085ae6L, 0xff0f6a70L, 0x66063bcaL, 0x11010b5cL,
		0x8f659effL, 0xf862ae69L, 0x616bffd3L, 0x166ccf45L, 0xa00ae278L,
		0xd70dd2eeL, 0x4e048354L, 0x3903b3c2L, 0xa7672661L, 0xd06016f7L,
		0x4969474dL, 0x3e6e77dbL, 0xaed16a4aL, 0xd9d65adcL, 0x40df0b66L,
		0x37d83bf0L, 0xa9bcae53L, 0xdebb9ec5L, 0x47b2cf7fL, 0x30b5ffe9L,
		0xbdbdf21cL, 0xcabac28aL, 0x53b39330L, 0x24b4a3a6L, 0xbad03605L,
		0xcdd70693L, 0x54de5729L, 0x23d967bfL, 0xb3667a2eL, 0xc4614ab8L,
		0x5d681b02L, 0x2a6f2b94L, 0xb40bbe37L, 0xc30c8ea1L, 0x5a05df1bL,
		0x2d02ef8dL
		};

#define DO1(buf) crc = crc_table[((int)crc ^ (*buf++)) & 0xff] ^ (crc >> 8);
#define DO2(buf)  DO1(buf); DO1(buf);
#define DO4(buf)  DO2(buf); DO2(buf);
#define DO8(buf)  DO4(buf); DO4(buf);

	/* ========================================================================= */

	uint32_t CUtils::computeCRC32 (uint8_t * buf, uint32_t len)
	{
		if ((buf == nullptr) || (len == 0))
			return 0;

		uint32_t crc = 0;

		crc = crc ^ 0xffffffffL;
		//	while (len >= 8)
		//	{
		//		DO8(buf);
		//		len -= 8;
		//	}
		if (len) do {
				DO1(buf);
			} while (--len);
		return crc ^ 0xffffffffL;

	}

	void CUtils::writeStringVariable(const std::string & sString, char * pVariable, uint32_t nCount)
	{
		int nIndex = 0;
		for (char ch : sString) {
			pVariable[nIndex] = ch;
			nIndex++;
			if ((nIndex + 1) >= nCount)
				break;
		}
		pVariable[nIndex] = 0;
	}

}
```

#### SignalHandler.hpp
```cpp
/*++

Copyright (C) 2024 Institute for Machine Tools and Industrial Management
TUM School of Engineering and Design
Technical University of Munich

All rights reserved.

Redistribution and use in source and binary forms, with or without
modification, are permitted provided that the following conditions are met:
	* Redistributions of source code must retain the above copyright
	  notice, this list of conditions and the following disclaimer.
	* Redistributions in binary form must reproduce the above copyright
	  notice, this list of conditions and the following disclaimer in the
	  documentation and/or other materials provided with the distribution.
	* Neither the name of the Technical University of Munich nor the
	  names of its contributors may be used to endorse or promote products
	  derived from this software without specific prior written permission.

THIS SOFTWARE IS PROVIDED BY THE COPYRIGHT HOLDERS AND CONTRIBUTORS "AS IS" AND
ANY EXPRESS OR IMPLIED WARRANTIES, INCLUDING, BUT NOT LIMITED TO, THE IMPLIED
WARRANTIES OF MERCHANTABILITY AND FITNESS FOR A PARTICULAR PURPOSE ARE
DISCLAIMED. IN NO EVENT SHALL TECHNICAL UNIVERSITY OF MUNICH BE LIABLE FOR ANY
DIRECT, INDIRECT, INCIDENTAL, SPECIAL, EXEMPLARY, OR CONSEQUENTIAL DAMAGES
(INCLUDING, BUT NOT LIMITED TO, PROCUREMENT OF SUBSTITUTE GOODS OR SERVICES;
LOSS OF USE, DATA, OR PROFITS; OR BUSINESS INTERRUPTION) HOWEVER CAUSED AND
ON ANY THEORY OF LIABILITY, WHETHER IN CONTRACT, STRICT LIABILITY, OR TORT
(INCLUDING NEGLIGENCE OR OTHERWISE) ARISING IN ANY WAY OUT OF THE USE OF THIS
SOFTWARE, EVEN IF ADVISED OF THE POSSIBILITY OF SUCH DAMAGE.

*/

#ifndef __SIGNALHANDLER_HPP
#define __SIGNALHANDLER_HPP

#include "Framework.hpp"
#include "SystemInfo.hpp"
#include <queue>

namespace BuRCPP {

	enum class eSignalParameterType : int32_t {
		UnknownParameterType = 0,
		BoolParameterType = 1,
		Int32ParameterType = 2,
		Uint32ParameterType = 3,
		DoubleParameterType = 4
	};

	class CSignalSendInstance;
	class CSignalProcessingInstance;
	class CSignalDefinition;
	class CSignalInstanceBase;

	class CSignalParameterDefinition {

		private:

		std::string m_sName;
		uint32_t m_nMemoryAddress;

		public:

		CSignalParameterDefinition (const std::string & sName, uint32_t nMemoryAddress);
		virtual ~CSignalParameterDefinition ();

		std::string getName ();

		uint32_t getMemoryAddress () const;
		virtual eSignalParameterType getSignalType () = 0;
		virtual uint32_t getSizeInBytes () = 0;

		virtual void writeDefaultToInstance (CSignalInstanceBase * pInstance) = 0;

		virtual void writeIntegerToInstance (CSignalInstanceBase * pInstance, int64_t nValue);
		virtual void writeDoubleToInstance (CSignalInstanceBase * pInstance, double dValue);
		virtual int64_t readIntegerFromInstance (CSignalInstanceBase * pInstance);
		virtual double readDoubleFromInstance (CSignalInstanceBase * pInstance);
	};

	class CSignalBoolParameterDefinition : public CSignalParameterDefinition {
		private:
		bool m_bDefaultValue;

		public:

		CSignalBoolParameterDefinition (const std::string & sName, uint32_t nMemoryAddress, bool bDefaultValue);
		virtual ~CSignalBoolParameterDefinition ();
		virtual eSignalParameterType getSignalType () override;
		virtual uint32_t getSizeInBytes () override;

		virtual void writeDefaultToInstance (CSignalInstanceBase * pInstance) override;
		virtual void writeIntegerToInstance (CSignalInstanceBase * pInstance, int64_t nValue) override;
		virtual int64_t readIntegerFromInstance (CSignalInstanceBase * pInstance) override;
	};

	class CSignalInt32ParameterDefinition : public CSignalParameterDefinition {
		private:
		int32_t m_nDefaultValue;
		public:

		CSignalInt32ParameterDefinition (const std::string & sName, uint32_t nMemoryAddress, int32_t nDefaultValue);
		virtual ~CSignalInt32ParameterDefinition ();
		virtual eSignalParameterType getSignalType () override;
		virtual uint32_t getSizeInBytes () override;

		virtual void writeDefaultToInstance (CSignalInstanceBase * pInstance) override;
		virtual void writeIntegerToInstance (CSignalInstanceBase * pInstance, int64_t nValue) override;
		virtual int64_t readIntegerFromInstance (CSignalInstanceBase * pInstance) override;

	};

	class CSignalUint32ParameterDefinition : public CSignalParameterDefinition {
		private:
		uint32_t m_nDefaultValue;
		public:

		CSignalUint32ParameterDefinition (const std::string & sName, uint32_t nMemoryAddress, uint32_t nDefaultValue);
		virtual ~CSignalUint32ParameterDefinition ();
		virtual eSignalParameterType getSignalType () override;
		virtual uint32_t getSizeInBytes () override;

		virtual void writeDefaultToInstance (CSignalInstanceBase * pInstance) override;
		virtual void writeIntegerToInstance (CSignalInstanceBase * pInstance, int64_t nValue) override;
		virtual int64_t readIntegerFromInstance (CSignalInstanceBase * pInstance) override;

	};

	class CSignalFloatParameterDefinition : public CSignalParameterDefinition {
		private:
		float m_fDefaultValue;
		public:

		CSignalFloatParameterDefinition (const std::string & sName, uint32_t nMemoryAddress, float fDefaultValue);
		virtual ~CSignalFloatParameterDefinition ();
		virtual eSignalParameterType getSignalType () override;
		virtual uint32_t getSizeInBytes () override;

		virtual void writeDefaultToInstance (CSignalInstanceBase * pInstance) override;
		virtual void writeDoubleToInstance (CSignalInstanceBase * pInstance, double dValue) override;
		virtual double readDoubleFromInstance (CSignalInstanceBase * pInstance) override;

	};

	class CSignalDoubleParameterDefinition : public CSignalParameterDefinition {
		private:
		double m_dDefaultValue;
		public:

		CSignalDoubleParameterDefinition (const std::string & sName, uint32_t nMemoryAddress, double dDefaultValue);
		virtual ~CSignalDoubleParameterDefinition ();
		virtual eSignalParameterType getSignalType () override;
		virtual uint32_t getSizeInBytes () override;

		virtual void writeDefaultToInstance (CSignalInstanceBase * pInstance) override;
		virtual void writeDoubleToInstance (CSignalInstanceBase * pInstance, double dValue) override;
		virtual double readDoubleFromInstance (CSignalInstanceBase * pInstance) override;

	};

	class CSignalInstanceBase {
		protected:

		CSignalDefinition* m_pDefinition;
		uint32_t m_nInstanceID;

		uint8_t * m_pMemory;
		uint32_t m_nMemorySize;

		public:

		CSignalInstanceBase	(CSignalDefinition* pDefinition, uint32_t nInstanceID, uint8_t * pMemory, uint32_t nMemorySize);

		virtual ~CSignalInstanceBase ();

		void writeData (uint8_t * pSource, uint32_t nOffset, uint32_t nSize);
		void readData (uint8_t * pTarget, uint32_t nOffset, uint32_t nSize);

		bool signalHasBeenProcessed ();

		bool getBoolParameter (const std::string & sName);
		int32_t getInt32Parameter (const std::string & sName);
		uint32_t getUint32Parameter (const std::string & sName);
		double getDoubleParameter (const std::string & sName);
		float getFloatParameter (const std::string & sName);

		bool getBoolResult (const std::string & sName);
		int32_t getInt32Result (const std::string & sName);
		uint32_t getUint32Result (const std::string & sName);
		double getDoubleResult (const std::string & sName);
		float getFloatResult (const std::string & sName);

		bool signalIsTriggered ();

		uint32_t getInstanceID ();

	};

	class CSignalProcessingInstance : public CSignalInstanceBase {

		public:

		CSignalProcessingInstance (CSignalDefinition* pDefinition, uint32_t nInstanceID, uint8_t * pMemory, uint32_t nMemorySize);
		virtual ~CSignalProcessingInstance ();

		void setBoolResult (const std::string & sName, bool bValue);
		void setInt32Result (const std::string & sName, int32_t nValue);
		void setUint32Result (const std::string & sName, uint32_t nValue);
		void setDoubleResult (const std::string & sName, double dValue);
		void setFloatResult (const std::string & sName, float fValue);

		void finishProcessing ();

	};

	class CSignalSendInstance : public CSignalInstanceBase {
		private:

			uint64_t m_nTriggerTimeInMicroseconds;

		public:

		CSignalSendInstance (CSignalDefinition* pDefinition, uint32_t nInstanceID, uint8_t * pMemory, uint32_t nMemorySize);
		virtual ~CSignalSendInstance ();

		void setBoolParameter (const std::string & sName, bool bValue);
		void setInt32Parameter (const std::string & sName, int32_t nValue);
		void setUint32Parameter (const std::string & sName, uint32_t nValue);
		void setDoubleParameter (const std::string & sName, double dValue);
		void setFloatParameter (const std::string & sName, float fValue);

		bool triggerSignal ();

		void resetTriggerTime ();
		uint64_t getTriggerTimeInMicroseconds ();

	};

	class CSignalInstance : public CSignalInstanceBase {
		private:

		std::shared_ptr<CSignalSendInstance> m_SendInstance;
		std::shared_ptr<CSignalProcessingInstance> m_ProcessingInstance;
		public:

		CSignalInstance (CSignalDefinition* pDefinition, uint32_t nInstanceID, uint8_t * pMemory, uint32_t nMemorySize);
		virtual ~CSignalInstance ();

		std::shared_ptr<CSignalSendInstance> getSendInstance ();
		std::shared_ptr<CSignalProcessingInstance> getProcessingInstance ();

		bool signalLifeTimeIsExpired ();
		void resetTimer ();
	};

	class CSignalDefinition {
		private:

		uint32_t m_nLifeTimeInMilliseconds;
		std::shared_ptr<CSystemInfo> m_pSystemInfo;

		std::string m_sName;
		uint32_t m_nQueueSize;
		std::map<std::string, std::shared_ptr<CSignalParameterDefinition>> m_Parameters;
		std::map<std::string, std::shared_ptr<CSignalParameterDefinition>> m_Results;

		std::vector<uint8_t> m_MemoryBuffer;
		uint32_t m_nCurrentMemorySizePerInstance;

		std::map<uint32_t, std::shared_ptr<CSignalInstance>> m_Instances;
		std::queue<std::shared_ptr<CSignalInstance>> m_UnusedInstanceQueue;
		std::map<uint32_t, std::shared_ptr<CSignalInstance>> m_InPreparationInstanceQueue;
		std::queue<std::shared_ptr<CSignalInstance>> m_ActiveInstanceQueue;
		std::map<uint32_t, std::shared_ptr<CSignalInstance>> m_InProcessInstanceQueue;
		std::queue<std::shared_ptr<CSignalInstance>> m_FinishedInstanceQueue;

		bool isInitializing ();

		void registerParameter (std::shared_ptr<CSignalParameterDefinition> pParameter);
		void registerResult (std::shared_ptr<CSignalParameterDefinition> pResult);

		public:

		CSignalDefinition (const std::string & sName, const uint32_t nQueueSize, const uint32_t nLifeTimeInMilliseconds, std::shared_ptr<CSystemInfo> pSystemInfo);
		virtual ~CSignalDefinition ();

		std::string getName ();

		void addBoolParameter (const std::string & sName, bool bDefault);
		void addInt32Parameter (const std::string & sName, int32_t nDefault);
		void addUint32Parameter (const std::string & sName, uint32_t nDefault);
		void addDoubleParameter (const std::string & sName, double dDefault);

		void addBoolResult (const std::string & sName, bool bDefault);
		void addInt32Result (const std::string & sName, int32_t nDefault);
		void addUint32Result (const std::string & sName, uint32_t nDefault);
		void addDoubleResult (const std::string & sName, double dDefault);

		void buildInstances ();

		CSignalParameterDefinition * findParameter (const std::string & sName, bool bMustExist);
		CSignalParameterDefinition * findResult (const std::string & sName, bool bMustExist);

		CSignalSendInstance * prepareSignal ();
		CSignalProcessingInstance * checkSignal ();

		void finishPreparation (CSignalSendInstance * pSignalInstance);
		void finishProcessing (CSignalProcessingInstance * pSignalInstance);

		uint32_t getLifeTimeInMilliseconds ();
		uint64_t getSystemTimeInMicroseconds ();

		bool signalLifeTimeIsExpired (CSignalSendInstance * pSignalInstance);
		void releaseExpiredSignals ();

	};

	class CSignalHandler {

		private:

		std::shared_ptr<CSystemInfo> m_pSystemInfo;

		std::map<std::string, std::shared_ptr<CSignalDefinition>> m_SignalDefinitions;

		bool m_bIsInitializing;

		public:

		CSignalHandler (std::shared_ptr<CSystemInfo> pSystemInfo);

		virtual ~CSignalHandler ();

		std::shared_ptr<CSignalDefinition> registerSignal (const std::string & sName, const uint32_t nQueueSize, const uint32_t nLifetimeInMilliseconds);

		CSignalProcessingInstance * checkSignal (const std::string & sName);
		CSignalSendInstance * prepareSignal (const std::string & sName);

		void buildInstances ();

		void releaseExpiredSignals ();

	};

};

#endif
```

#### SignalHandler.cpp
```cpp
/*++

Copyright (C) 2024 Institute for Machine Tools and Industrial Management
TUM School of Engineering and Design
Technical University of Munich

All rights reserved.

Redistribution and use in source and binary forms, with or without
modification, are permitted provided that the following conditions are met:
	* Redistributions of source code must retain the above copyright
	  notice, this list of conditions and the following disclaimer.
	* Redistributions in binary form must reproduce the above copyright
	  notice, this list of conditions and the following disclaimer in the
	  documentation and/or other materials provided with the distribution.
	* Neither the name of the Technical University of Munich nor the
	  names of its contributors may be used to endorse or promote products
	  derived from this software without specific prior written permission.

THIS SOFTWARE IS PROVIDED BY THE COPYRIGHT HOLDERS AND CONTRIBUTORS "AS IS" AND
ANY EXPRESS OR IMPLIED WARRANTIES, INCLUDING, BUT NOT LIMITED TO, THE IMPLIED
WARRANTIES OF MERCHANTABILITY AND FITNESS FOR A PARTICULAR PURPOSE ARE
DISCLAIMED. IN NO EVENT SHALL TECHNICAL UNIVERSITY OF MUNICH BE LIABLE FOR ANY
DIRECT, INDIRECT, INCIDENTAL, SPECIAL, EXEMPLARY, OR CONSEQUENTIAL DAMAGES
(INCLUDING, BUT NOT LIMITED TO, PROCUREMENT OF SUBSTITUTE GOODS OR SERVICES;
LOSS OF USE, DATA, OR PROFITS; OR BUSINESS INTERRUPTION) HOWEVER CAUSED AND
ON ANY THEORY OF LIABILITY, WHETHER IN CONTRACT, STRICT LIABILITY, OR TORT
(INCLUDING NEGLIGENCE OR OTHERWISE) ARISING IN ANY WAY OUT OF THE USE OF THIS
SOFTWARE, EVEN IF ADVISED OF THE POSSIBILITY OF SUCH DAMAGE.

*/

#include "SignalHandler.hpp"
#include "Utils.hpp"

#include <cstdint>
#include <limits>

#define SIGNALDEFINITION_MINQUEUESIZE 1
#define SIGNALDEFINITION_MAXQUEUESIZE 64

namespace BuRCPP
{

	CSignalParameterDefinition::CSignalParameterDefinition (const std::string & sName, uint32_t nMemoryAddress)
		: m_sName (sName), m_nMemoryAddress (nMemoryAddress)
	{
	}

	CSignalParameterDefinition::~CSignalParameterDefinition ()
	{
	}

	std::string CSignalParameterDefinition::getName ()
	{
		return m_sName;
	}

	uint32_t CSignalParameterDefinition::getMemoryAddress () const
	{
		return m_nMemoryAddress;
	}

	void CSignalParameterDefinition::writeIntegerToInstance (CSignalInstanceBase * pInstance, int64_t nValue)
	{
		throw CException (eErrorCode::COULDNOTWRITEINTEGERTOPARAMETER, "could not write integer value to signal parameter:." + m_sName);
	}

	void CSignalParameterDefinition::writeDoubleToInstance (CSignalInstanceBase * pInstance, double dValue)
	{
		throw CException (eErrorCode::COULDNOTWRITEDOUBLETOPARAMETER, "could not write double value to signal parameter:." + m_sName);
	}

	int64_t CSignalParameterDefinition::readIntegerFromInstance (CSignalInstanceBase * pInstance)
	{
		throw CException (eErrorCode::COULDNOTREADINTEGERFROMPARAMETER, "could not read integer value from signal parameter:." + m_sName);
	}

	double CSignalParameterDefinition::readDoubleFromInstance (CSignalInstanceBase * pInstance)
	{
		throw CException (eErrorCode::COULDNOTREADDOUBLEFROMPARAMETER, "could not read double value from signal parameter:." + m_sName);
	}

	CSignalBoolParameterDefinition::CSignalBoolParameterDefinition (const std::string & sName, uint32_t nMemoryAddress, bool bDefaultValue)
		: CSignalParameterDefinition (sName, nMemoryAddress), m_bDefaultValue (bDefaultValue)
	{
	}

	CSignalBoolParameterDefinition::~CSignalBoolParameterDefinition ()
	{
	}

	eSignalParameterType CSignalBoolParameterDefinition::getSignalType ()
	{
		return eSignalParameterType::BoolParameterType;
	}

	uint32_t CSignalBoolParameterDefinition::getSizeInBytes ()
	{
		return sizeof (uint8_t);
	}

	void CSignalBoolParameterDefinition::writeDefaultToInstance (CSignalInstanceBase * pInstance)
	{
		if (m_bDefaultValue)
			writeIntegerToInstance (pInstance,  1);
		else
			writeIntegerToInstance (pInstance,  0);
	}

	void CSignalBoolParameterDefinition::writeIntegerToInstance (CSignalInstanceBase * pInstance, int64_t nValue)
	{
		if (pInstance == nullptr)
			throw CException (eErrorCode::INVALIDPARAM, "invalid instance parameter");

		uint8_t nValueToWrite = 0;
		if (nValue != 0)
			nValueToWrite = 1;

		pInstance->writeData (&nValueToWrite, getMemoryAddress (), 1);

	}

	int64_t CSignalBoolParameterDefinition::readIntegerFromInstance (CSignalInstanceBase * pInstance)
	{
		if (pInstance == nullptr)
			throw CException (eErrorCode::INVALIDPARAM, "invalid instance parameter");

		uint8_t nReadValue = 0;
		pInstance->readData (&nReadValue, getMemoryAddress (), 1);

		if (nReadValue != 0)
			return 1;
		else
			return 0;

	}

	CSignalInt32ParameterDefinition::CSignalInt32ParameterDefinition (const std::string & sName, uint32_t nMemoryAddress, int32_t nDefaultValue)
		: CSignalParameterDefinition (sName, nMemoryAddress), m_nDefaultValue (nDefaultValue)
	{
	}

	CSignalInt32ParameterDefinition::~CSignalInt32ParameterDefinition ()
	{
	}

	eSignalParameterType CSignalInt32ParameterDefinition::getSignalType ()
	{
		return eSignalParameterType::Int32ParameterType;
	}

	uint32_t CSignalInt32ParameterDefinition::getSizeInBytes ()
	{
		return sizeof (int32_t);
	}

	void CSignalInt32ParameterDefinition::writeDefaultToInstance (CSignalInstanceBase * pInstance)
	{
		writeIntegerToInstance (pInstance,  m_nDefaultValue);
	}

	void CSignalInt32ParameterDefinition::writeIntegerToInstance (CSignalInstanceBase * pInstance, int64_t nValue)
	{
		if (pInstance == nullptr)
			throw CException (eErrorCode::INVALIDPARAM, "invalid instance parameter");

		if ((nValue < std::numeric_limits<std::int32_t>::min ()) || (nValue > std::numeric_limits<std::int32_t>::max ()))
			throw CException (eErrorCode::VALUEISOUTSIDEOFINTEGER32RANGE, "value is outside of integer 32 range: " + getName ());

		int32_t nValueToWrite = (int32_t) nValue;
		pInstance->writeData ((uint8_t*) &nValueToWrite, getMemoryAddress (), sizeof (int32_t));

	}

	int64_t CSignalInt32ParameterDefinition::readIntegerFromInstance (CSignalInstanceBase * pInstance)
	{
		if (pInstance == nullptr)
			throw CException (eErrorCode::INVALIDPARAM, "invalid instance parameter");

		int32_t nReadValue = 0;
		pInstance->readData ((uint8_t*)&nReadValue, getMemoryAddress (), sizeof (int32_t));

		return nReadValue;
	}

	CSignalUint32ParameterDefinition::CSignalUint32ParameterDefinition (const std::string & sName, uint32_t nMemoryAddress, uint32_t nDefaultValue)
		: CSignalParameterDefinition (sName, nMemoryAddress), m_nDefaultValue (nDefaultValue)
	{
	}

	CSignalUint32ParameterDefinition::~CSignalUint32ParameterDefinition ()
	{
	}

	eSignalParameterType CSignalUint32ParameterDefinition::getSignalType ()
	{
		return eSignalParameterType::Uint32ParameterType;
	}

	uint32_t CSignalUint32ParameterDefinition::getSizeInBytes ()
	{
		return sizeof (uint32_t);
	}

	void CSignalUint32ParameterDefinition::writeDefaultToInstance (CSignalInstanceBase * pInstance)
	{
		writeIntegerToInstance (pInstance,  m_nDefaultValue);
	}

	void CSignalUint32ParameterDefinition::writeIntegerToInstance (CSignalInstanceBase * pInstance, int64_t nValue)
	{
		if (pInstance == nullptr)
			throw CException (eErrorCode::INVALIDPARAM, "invalid instance parameter");

		if ((nValue < std::numeric_limits<std::uint32_t>::min ()) || (nValue > std::numeric_limits<std::uint32_t>::max ()))
			throw CException (eErrorCode::VALUEISOUTSIDEOFUNSIGNEDINTEGER32RANGE, "value is outside of unsigned integer 32 range: " + getName ());

		int32_t nValueToWrite = (int32_t) nValue;
		pInstance->writeData ((uint8_t*) &nValueToWrite, getMemoryAddress (), sizeof (int32_t));

	}

	int64_t CSignalUint32ParameterDefinition::readIntegerFromInstance (CSignalInstanceBase * pInstance)
	{
		if (pInstance == nullptr)
			throw CException (eErrorCode::INVALIDPARAM, "invalid instance parameter");

		int32_t nReadValue = 0;
		pInstance->readData ((uint8_t*)&nReadValue, getMemoryAddress (), sizeof (uint32_t));

		return nReadValue;
	}

	CSignalDoubleParameterDefinition::CSignalDoubleParameterDefinition (const std::string & sName, uint32_t nMemoryAddress, double dDefaultValue)
		: CSignalParameterDefinition (sName, nMemoryAddress), m_dDefaultValue (dDefaultValue)
	{
	}

	CSignalDoubleParameterDefinition::~CSignalDoubleParameterDefinition ()
	{
	}

	eSignalParameterType CSignalDoubleParameterDefinition::getSignalType ()
	{
		return eSignalParameterType::DoubleParameterType;
	}

	uint32_t CSignalDoubleParameterDefinition::getSizeInBytes ()
	{
		return sizeof (double);
	}

	void CSignalDoubleParameterDefinition::writeDefaultToInstance (CSignalInstanceBase * pInstance)
	{
		writeDoubleToInstance (pInstance,  m_dDefaultValue);
	}

	void CSignalDoubleParameterDefinition::writeDoubleToInstance (CSignalInstanceBase * pInstance, double dValue)
	{
		if (pInstance == nullptr)
			throw CException (eErrorCode::INVALIDPARAM, "invalid instance parameter");

		pInstance->writeData ((uint8_t*) &dValue, getMemoryAddress (), sizeof (dValue));

	}

	double CSignalDoubleParameterDefinition::readDoubleFromInstance (CSignalInstanceBase * pInstance)
	{
		if (pInstance == nullptr)
			throw CException (eErrorCode::INVALIDPARAM, "invalid instance parameter");

		double dReadValue = 0.0;
		pInstance->readData ((uint8_t*)&dReadValue, getMemoryAddress (), sizeof (double));

		return dReadValue;
	}

	CSignalDefinition::CSignalDefinition (const std::string & sName, const uint32_t nQueueSize, const uint32_t nLifeTimeInMilliseconds, std::shared_ptr<CSystemInfo> pSystemInfo)
		: m_sName (sName), m_nQueueSize (nQueueSize), m_nCurrentMemorySizePerInstance (0), m_nLifeTimeInMilliseconds (nLifeTimeInMilliseconds), m_pSystemInfo (pSystemInfo)
	{
		if (pSystemInfo.get () == nullptr)
			throw CException (eErrorCode::INVALIDPARAM, "invalid system info parameter");

		if ((nQueueSize < SIGNALDEFINITION_MINQUEUESIZE) || (nQueueSize > SIGNALDEFINITION_MAXQUEUESIZE))
			throw CException (eErrorCode::INVALIDSIGNALQUEUESIZE, "invalid signal queue size.");

		addBoolParameter ("__active", false);
		addBoolResult ("__processed", false);
	}

	CSignalDefinition::~CSignalDefinition ()
	{
	}

	std::string CSignalDefinition::getName ()
	{
		return m_sName;
	}

	bool CSignalDefinition::isInitializing ()
	{
		return (m_Instances.empty ());
	}

	void CSignalDefinition::registerParameter (std::shared_ptr<CSignalParameterDefinition> pParameter)
	{
		if (pParameter.get () == nullptr)
			throw CException (eErrorCode::INVALIDPARAM, "invalid signal parameter instance.");

		if (!isInitializing ())
			throw CException (eErrorCode::CANNOTREGISTERPARAMETER, "signal parameters can only be registered initialization mode.");

		if (pParameter->getMemoryAddress () != m_nCurrentMemorySizePerInstance)
			throw CException (eErrorCode::SIGNALMEMORYALLOCATIONERROR, "signal memory allocation error.");

		std::string sName = pParameter->getName ();
		auto iIter = m_Parameters.find (sName);
		if (iIter != m_Parameters.end ())
			throw CException (eErrorCode::DUPLICATESIGNALPARAMETERNAME, "duplicate signal parameter name: " + sName);

		m_Parameters.insert (std::make_pair (sName, pParameter));

		m_nCurrentMemorySizePerInstance += pParameter->getSizeInBytes ();

	}

	void CSignalDefinition::registerResult (std::shared_ptr<CSignalParameterDefinition> pResult)
	{
		if (pResult.get () == nullptr)
			throw CException (eErrorCode::INVALIDPARAM, "invalid signal result instance.");

		if (!isInitializing ())
			throw CException (eErrorCode::CANNOTREGISTERRESULT, "signal results can only be registered initialization mode.");

		if (pResult->getMemoryAddress () != m_nCurrentMemorySizePerInstance)
			throw CException (eErrorCode::SIGNALMEMORYALLOCATIONERROR, "signal memory allocation error.");

		std::string sName = pResult->getName ();
		auto iIter = m_Results.find (sName);
		if (iIter != m_Results.end ())
			throw CException (eErrorCode::DUPLICATESIGNALRESULTNAME, "duplicate signal result name: " + sName);

		m_Results.insert (std::make_pair (sName, pResult));

		m_nCurrentMemorySizePerInstance += pResult->getSizeInBytes ();

	}

	void CSignalDefinition::addBoolParameter (const std::string & sName, bool bDefault)
	{
		registerParameter (std::make_shared<CSignalBoolParameterDefinition> (sName, m_nCurrentMemorySizePerInstance, bDefault));
	}

	void CSignalDefinition::addInt32Parameter (const std::string & sName, int32_t nDefault)
	{
		registerParameter (std::make_shared<CSignalInt32ParameterDefinition> (sName, m_nCurrentMemorySizePerInstance, nDefault));

	}

	void CSignalDefinition::addUint32Parameter (const std::string & sName, uint32_t nDefault)
	{
		registerParameter (std::make_shared<CSignalUint32ParameterDefinition> (sName, m_nCurrentMemorySizePerInstance, nDefault));
	}

	void CSignalDefinition::addDoubleParameter (const std::string & sName, double dDefault)
	{
		registerParameter (std::make_shared<CSignalDoubleParameterDefinition> (sName, m_nCurrentMemorySizePerInstance, dDefault));
	}

	void CSignalDefinition::addBoolResult (const std::string & sName, bool bDefault)
	{
		registerResult (std::make_shared<CSignalBoolParameterDefinition> (sName, m_nCurrentMemorySizePerInstance, bDefault));
	}

	void CSignalDefinition::addInt32Result (const std::string & sName, int32_t nDefault)
	{
		registerResult (std::make_shared<CSignalInt32ParameterDefinition> (sName, m_nCurrentMemorySizePerInstance, nDefault));
	}

	void CSignalDefinition::addUint32Result (const std::string & sName, uint32_t nDefault)
	{
		registerResult (std::make_shared<CSignalUint32ParameterDefinition> (sName, m_nCurrentMemorySizePerInstance, nDefault));
	}

	void CSignalDefinition::addDoubleResult (const std::string & sName, double dDefault)
	{
		registerResult (std::make_shared<CSignalDoubleParameterDefinition> (sName, m_nCurrentMemorySizePerInstance, dDefault));
	}

	void CSignalDefinition::buildInstances ()
	{
		if (!isInitializing ())
			throw CException (eErrorCode::SIGNALINSTANCESALREADYBUILT, "signal instances have benn already built");

		m_MemoryBuffer.resize (m_nCurrentMemorySizePerInstance * m_nQueueSize);

		for (uint32_t nIndex = 0; nIndex < m_nQueueSize; nIndex++) {

			auto pSignal = std::make_shared<CSignalInstance> (this, nIndex + 1, &m_MemoryBuffer.at (nIndex * m_nCurrentMemorySizePerInstance), m_nCurrentMemorySizePerInstance);
			m_Instances.insert (std::make_pair(pSignal->getInstanceID (), pSignal));
			m_UnusedInstanceQueue.push (pSignal);

		}

	}

	CSignalParameterDefinition * CSignalDefinition::findParameter (const std::string & sName, bool bMustExist)
	{
		auto iIter = m_Parameters.find (sName);
		if (iIter == m_Parameters.end ()) {
			if (bMustExist)
				throw CException (eErrorCode::SIGNALPARAMETERNOTFOUND, "signal parameter not found: " + sName);

			return nullptr;
		}

		return iIter->second.get ();
	}

	CSignalSendInstance * CSignalDefinition::prepareSignal ()
	{

		if (m_Instances.size () == 0)
			throw CException (eErrorCode::SIGNALHASNOINSTANCES, "signal has no instances: " + m_sName);

		if (m_UnusedInstanceQueue.empty ())
			throw CException (eErrorCode::COULDNOTPREPARESIGNAL, "signal instances queue is full: " + m_sName);

		auto pSignal = m_UnusedInstanceQueue.front ();
		m_UnusedInstanceQueue.pop ();
		m_InPreparationInstanceQueue.insert (std::make_pair (pSignal->getInstanceID (), pSignal));

		pSignal->resetTimer ();

		for (auto pParameter: m_Parameters)
			pParameter.second->writeDefaultToInstance (pSignal.get ());
		for (auto pResult: m_Results)
			pResult.second->writeDefaultToInstance (pSignal.get ());

		return pSignal->getSendInstance ().get ();

	}

	CSignalProcessingInstance * CSignalDefinition::checkSignal ()
	{
		if (m_Instances.size () == 0)
			throw CException (eErrorCode::SIGNALHASNOINSTANCES, "signal has no instances: " + m_sName);

		if (m_ActiveInstanceQueue.empty ())
			return nullptr;

		auto pSignal = m_ActiveInstanceQueue.front ();
		m_ActiveInstanceQueue.pop ();
		m_InProcessInstanceQueue.insert (std::make_pair (pSignal->getInstanceID (), pSignal));

		return pSignal->getProcessingInstance ().get ();

	}

	void CSignalDefinition::finishProcessing (CSignalProcessingInstance * pProcessingInstance)
	{
		if (m_Instances.size () == 0)
			throw CException (eErrorCode::SIGNALHASNOINSTANCES, "signal has no instances: " + m_sName);

		uint32_t nInstanceID = pProcessingInstance->getInstanceID();
		auto iIter = m_InProcessInstanceQueue.find (nInstanceID);
		if (iIter == m_InProcessInstanceQueue.end ())
			throw CException (eErrorCode::SIGNALISNOTINPROCESS, "signal is not in process" + m_sName);

		auto pSignal = iIter->second;
		m_InProcessInstanceQueue.erase (nInstanceID);

		pProcessingInstance->setBoolResult ("__processed", true);

		if (pSignal->signalLifeTimeIsExpired ()) {
			m_UnusedInstanceQueue.push (pSignal);
			pSignal->resetTimer ();
		} else {

			m_FinishedInstanceQueue.push (pSignal);
		}

	}

	void CSignalDefinition::releaseExpiredSignals ()
	{

		while (!m_FinishedInstanceQueue.empty ()) {
			auto pSignal = m_FinishedInstanceQueue.front ();
			if (pSignal->signalLifeTimeIsExpired ()) {
				m_FinishedInstanceQueue.pop ();
				m_UnusedInstanceQueue.push (pSignal);
				pSignal->resetTimer ();
			} else {
				break;
			}
		}

	}

	void CSignalDefinition::finishPreparation (CSignalSendInstance * pSignalInstance)
	{
		if (m_Instances.size () == 0)
			throw CException (eErrorCode::SIGNALHASNOINSTANCES, "signal has no instances: " + m_sName);

		uint32_t nInstanceID = pSignalInstance->getInstanceID();
		auto iIter = m_InPreparationInstanceQueue.find (nInstanceID);
		if (iIter == m_InPreparationInstanceQueue.end ())
			throw CException (eErrorCode::SIGNALISNOTINPREPARATION, "signal is not in preparation" + m_sName);

		auto pSignal = iIter->second;
		m_InPreparationInstanceQueue.erase (nInstanceID);
		m_ActiveInstanceQueue.push (pSignal);

		pSignalInstance->setBoolParameter ("__active", true);
	}

	CSignalParameterDefinition * CSignalDefinition::findResult (const std::string & sName, bool bMustExist)
	{
		auto iIter = m_Results.find (sName);
		if (iIter == m_Results.end ()) {
			if (bMustExist)
				throw CException (eErrorCode::SIGNALRESULTNOTFOUND, "signal result not found: " + sName);

			return nullptr;
		}

		return iIter->second.get ();
	}

	uint32_t CSignalDefinition::getLifeTimeInMilliseconds ()
	{
		return m_nLifeTimeInMilliseconds;
	}

	uint64_t CSignalDefinition::getSystemTimeInMicroseconds ()
	{
		return m_pSystemInfo->getSystemTimeInMicroseconds ();
	}

	CSignalInstanceBase::CSignalInstanceBase (CSignalDefinition* pDefinition, uint32_t nInstanceID, uint8_t * pMemory, uint32_t nMemorySize)
	: m_pDefinition (pDefinition), m_pMemory (pMemory), m_nMemorySize (nMemorySize), m_nInstanceID (nInstanceID)
	{
		if (pDefinition == nullptr)
			throw CException (eErrorCode::INVALIDPARAM, "invalid signal definition parameter");

		// ATTENTION: pMemory is allowed to be NULL!
		if (m_pMemory == nullptr) {
			if (m_nMemorySize != 0)
				throw CException (eErrorCode::INVALIDPARAM, "invalid memory size parameter");

		} else {
			if (m_nMemorySize == 0)
				throw CException (eErrorCode::INVALIDPARAM, "invalid memory size parameter");
		}

	}

	CSignalInstanceBase::~CSignalInstanceBase ()
	{

	}

	bool CSignalInstanceBase::signalHasBeenProcessed ()
	{
		return getBoolResult ("__processed");
	}

	void CSignalInstanceBase::writeData (uint8_t * pSource, uint32_t nOffset, uint32_t nSize)
	{
		if (nSize == 0)
			return;
		if (pSource == nullptr)
			throw CException (eErrorCode::INVALIDPARAM, "invalid signal parameter source data: " +  m_pDefinition->getName ());
		if (m_pMemory == nullptr)
			throw CException (eErrorCode::SIGNALDATAMISSINGMEMORY, "signal data is missing memory: " + m_pDefinition->getName ());

		if (nOffset >= m_nMemorySize)
			throw CException (eErrorCode::SIGNALDATAWRITEOUTOFRANGE, "signal data wanted to write out of range: " +  m_pDefinition->getName ());

		if ((nOffset + nSize) > m_nMemorySize)
			throw CException (eErrorCode::SIGNALDATAWRITEOUTOFRANGE, "signal data write exceeds buffer: " +  m_pDefinition->getName ());

		for (uint32_t nIndex = 0; nIndex < nSize; nIndex++)
			m_pMemory[nOffset + nIndex] = pSource[nIndex];
	}

	void CSignalInstanceBase::readData (uint8_t * pTarget, uint32_t nOffset, uint32_t nSize)
	{
		if (nSize == 0)
			return;
		if (pTarget == nullptr)
			throw CException (eErrorCode::INVALIDPARAM, "invalid signal parameter target data: " +  m_pDefinition->getName ());
		if (m_pMemory == nullptr)
			throw CException (eErrorCode::SIGNALDATAMISSINGMEMORY, "signal data is missing memory: " + m_pDefinition->getName ());

		if (nOffset >= m_nMemorySize)
			throw CException (eErrorCode::SIGNALDATAREADOUTOFRANGE, "signal data wanted to read out of range: " +  m_pDefinition->getName ());

		if ((nOffset + nSize) > m_nMemorySize)
			throw CException (eErrorCode::SIGNALDATAREADOUTOFRANGE, "signal data read exceeds buffer: " +  m_pDefinition->getName ());

		for (uint32_t nIndex = 0; nIndex < nSize; nIndex++)
			pTarget[nIndex] = m_pMemory[nOffset + nIndex];
	}

	CSignalProcessingInstance::CSignalProcessingInstance (CSignalDefinition* pDefinition, uint32_t nInstanceID, uint8_t * pMemory, uint32_t nMemorySize)
	  : CSignalInstanceBase (pDefinition, nInstanceID, pMemory, nMemorySize)
	{
		if (pDefinition == nullptr)
			throw CException (eErrorCode::INVALIDPARAM, "invalid signal definition variable");
	}

	CSignalProcessingInstance::~CSignalProcessingInstance ()
	{
	}

void CSignalProcessingInstance::setBoolResult (const std::string & sName, bool bValue)
{
	auto pResult = m_pDefinition->findResult (sName, true);
	if (bValue)
		pResult->writeIntegerToInstance (this, 1);
	else
		pResult->writeIntegerToInstance (this, 0);
}

void CSignalProcessingInstance::setInt32Result (const std::string & sName, int32_t nValue)
{
	auto pResult = m_pDefinition->findResult (sName, true);
	pResult->writeIntegerToInstance (this, (int64_t) nValue);
}

void CSignalProcessingInstance::setUint32Result (const std::string & sName, uint32_t nValue)
{
	auto pResult = m_pDefinition->findResult (sName, true);
	pResult->writeIntegerToInstance (this, (int64_t) nValue);
}

void CSignalProcessingInstance::setDoubleResult (const std::string & sName, double dValue)
{
	auto pResult = m_pDefinition->findResult (sName, true);
	pResult->writeDoubleToInstance (this, dValue);
}

void CSignalProcessingInstance::setFloatResult (const std::string & sName, float fValue)
{
	auto pResult = m_pDefinition->findResult (sName, true);
	pResult->writeDoubleToInstance (this, (double) fValue);
}

uint32_t CSignalInstanceBase::getInstanceID ()
{
	return m_nInstanceID;
}

bool CSignalInstanceBase::getBoolParameter (const std::string & sName)
{
	auto pParameter = m_pDefinition->findParameter (sName, true);
	int64_t nValue = pParameter->readIntegerFromInstance (this);

	return (nValue != 0);
}

int32_t CSignalInstanceBase::getInt32Parameter (const std::string & sName)
{
	auto pParameter = m_pDefinition->findParameter (sName, true);
	int64_t nValue = pParameter->readIntegerFromInstance (this);

	if ((nValue < std::numeric_limits<std::int32_t>::min ()) || (nValue > std::numeric_limits<std::int32_t>::max ()))
		throw CException (eErrorCode::VALUEISOUTSIDEOFINTEGER32RANGE, "value is outside of integer 32 range: " + sName);

	return (int32_t) nValue;

}

uint32_t CSignalInstanceBase::getUint32Parameter (const std::string & sName)
{
	auto pParameter = m_pDefinition->findParameter (sName, true);
	int64_t nValue = pParameter->readIntegerFromInstance (this);

	if ((nValue < std::numeric_limits<std::uint32_t>::min ()) || (nValue > std::numeric_limits<std::uint32_t>::max ()))
		throw CException (eErrorCode::VALUEISOUTSIDEOFUNSIGNEDINTEGER32RANGE, "value is outside of unsigned integer 32 range: " + sName);

	return (uint32_t) nValue;
}

double CSignalInstanceBase::getDoubleParameter (const std::string & sName)
{
	auto pParameter = m_pDefinition->findParameter (sName, true);
	return pParameter->readDoubleFromInstance (this);
}

float CSignalInstanceBase::getFloatParameter (const std::string & sName)
{
	auto pParameter = m_pDefinition->findParameter (sName, true);
	return (float) pParameter->readDoubleFromInstance (this);
}

bool CSignalInstanceBase::getBoolResult (const std::string & sName)
{
	auto pParameter = m_pDefinition->findResult (sName, true);
	int64_t nValue = pParameter->readIntegerFromInstance (this);

	return (nValue != 0);
}

int32_t CSignalInstanceBase::getInt32Result (const std::string & sName)
{
	auto pResult = m_pDefinition->findResult (sName, true);
	int64_t nValue = pResult->readIntegerFromInstance (this);

	if ((nValue < std::numeric_limits<std::int32_t>::min ()) || (nValue > std::numeric_limits<std::int32_t>::max ()))
		throw CException (eErrorCode::VALUEISOUTSIDEOFINTEGER32RANGE, "value is outside of integer 32 range: " + sName);

	return (int32_t) nValue;
}

uint32_t CSignalInstanceBase::getUint32Result (const std::string & sName)
{
	auto pResult = m_pDefinition->findResult (sName, true);
	int64_t nValue = pResult->readIntegerFromInstance (this);

	if ((nValue < std::numeric_limits<std::uint32_t>::min ()) || (nValue > std::numeric_limits<std::uint32_t>::max ()))
		throw CException (eErrorCode::VALUEISOUTSIDEOFUNSIGNEDINTEGER32RANGE, "value is outside of unsigned integer 32 range: " + sName);

	return (int32_t) nValue;
}

double CSignalInstanceBase::getDoubleResult (const std::string & sName)
{
	auto pResult = m_pDefinition->findResult (sName, true);
	return pResult->readDoubleFromInstance (this);

}

float CSignalInstanceBase::getFloatResult (const std::string & sName)
{
	auto pResult = m_pDefinition->findResult (sName, true);
	return (float) pResult->readDoubleFromInstance (this);

}

	void CSignalProcessingInstance::finishProcessing ()
	{
		m_pDefinition->finishProcessing (this);
	}

	CSignalSendInstance::CSignalSendInstance (CSignalDefinition* pDefinition, uint32_t nInstanceID, uint8_t * pMemory, uint32_t nMemorySize)
	: CSignalInstanceBase (pDefinition, nInstanceID, pMemory, nMemorySize), m_nTriggerTimeInMicroseconds (0)
	{
		if (pDefinition == nullptr)
			throw CException (eErrorCode::INVALIDPARAM, "invalid signal definition variable");
	}

	CSignalSendInstance::~CSignalSendInstance ()
	{
	}

	void CSignalSendInstance::resetTriggerTime ()
	{
		m_nTriggerTimeInMicroseconds = 0;
	}

void CSignalSendInstance::setBoolParameter (const std::string & sName, bool bValue)
{
	auto pParameter = m_pDefinition->findParameter (sName, true);
	if (bValue)
		pParameter->writeIntegerToInstance (this, 1);
	else
		pParameter->writeIntegerToInstance (this, 0);

}

void CSignalSendInstance::setInt32Parameter (const std::string & sName, int32_t nValue)
{
	auto pParameter = m_pDefinition->findParameter (sName, true);
	pParameter->writeIntegerToInstance (this, (int64_t) nValue);
}

void CSignalSendInstance::setUint32Parameter (const std::string & sName, uint32_t nValue)
{
	auto pParameter = m_pDefinition->findParameter (sName, true);
	pParameter->writeIntegerToInstance (this, (int64_t) nValue);
}

void CSignalSendInstance::setDoubleParameter (const std::string & sName, double dValue)
{
	auto pParameter = m_pDefinition->findParameter (sName, true);
	pParameter->writeDoubleToInstance (this, dValue);
}

void CSignalSendInstance::setFloatParameter (const std::string & sName, float fValue)
{
	auto pParameter = m_pDefinition->findParameter (sName, true);
	pParameter->writeDoubleToInstance (this, (double)fValue);
}

	bool CSignalInstanceBase::signalIsTriggered ()
	{
		return getBoolParameter ("__active");
	}

	bool CSignalSendInstance::triggerSignal ()
	{
		m_pDefinition->finishPreparation (this);

		m_nTriggerTimeInMicroseconds = m_pDefinition->getSystemTimeInMicroseconds ();

		return true;

	}

	uint64_t CSignalSendInstance::getTriggerTimeInMicroseconds ()
	{
		return m_nTriggerTimeInMicroseconds;
	}

	CSignalInstance::CSignalInstance (CSignalDefinition* pDefinition, uint32_t nInstanceID, uint8_t * pMemory, uint32_t nMemorySize)
	:  CSignalInstanceBase (pDefinition, nInstanceID, pMemory, nMemorySize)
	{
		m_SendInstance = std::make_shared<CSignalSendInstance> (pDefinition, getInstanceID(), pMemory, nMemorySize);
		m_ProcessingInstance = std::make_shared<CSignalProcessingInstance> (pDefinition, getInstanceID(),pMemory, nMemorySize);
	}

	CSignalInstance::~CSignalInstance ()
	{
	}

	std::shared_ptr<CSignalSendInstance> CSignalInstance::getSendInstance ()
	{
		return m_SendInstance;
	}

	std::shared_ptr<CSignalProcessingInstance> CSignalInstance::getProcessingInstance ()
	{
		return m_ProcessingInstance;
	}

	void CSignalInstance::resetTimer ()
	{
		m_SendInstance->resetTriggerTime();
	}

	bool CSignalInstance::signalLifeTimeIsExpired ()
	{
		uint64_t nTriggerTimeInMicroseconds = m_SendInstance->getTriggerTimeInMicroseconds ();
		uint64_t nCurrentTimeInMicroseconds = m_pDefinition->getSystemTimeInMicroseconds ();

		if (nCurrentTimeInMicroseconds >= nTriggerTimeInMicroseconds) {

			uint64_t nSignalExistenceTimeInMicroseconds = nCurrentTimeInMicroseconds - nTriggerTimeInMicroseconds;
			uint64_t nSignalExistenceTimeInMilliseconds = nSignalExistenceTimeInMicroseconds / 1000;

			return (nSignalExistenceTimeInMilliseconds > m_pDefinition->getLifeTimeInMilliseconds ());

		} else {
			throw CException (eErrorCode::SIGNALTRIGGERTIMEISINFUTURE, "signal trigger time is in the future");
		}

	}

CSignalHandler::CSignalHandler (std::shared_ptr<CSystemInfo> pSystemInfo)
	: m_bIsInitializing (true), m_pSystemInfo (pSystemInfo)
{
	if (pSystemInfo.get () == nullptr)
		throw CException (eErrorCode::INVALIDPARAM, "invalid system info parameter");
}

CSignalHandler::~CSignalHandler ()
{
}

std::shared_ptr<CSignalDefinition> CSignalHandler::registerSignal (const std::string & sName, const uint32_t nQueueSize, const uint32_t nLifetimeInMilliseconds)
{
	if (m_bIsInitializing) {

		auto iIter = m_SignalDefinitions.find (sName);
		if (iIter != m_SignalDefinitions.end ())
			throw CException (eErrorCode::DUPLICATESIGNALDEFINITION, "duplicate signal definition: " + sName);

		auto pSignalDefinition = std::make_shared<CSignalDefinition> (sName, nQueueSize, nLifetimeInMilliseconds, m_pSystemInfo);
		m_SignalDefinitions.insert (std::make_pair (sName, pSignalDefinition));

		return pSignalDefinition;

	} else {
		throw CException (eErrorCode::CANNOTREGISTERSIGNAL, "can not register signal, if not in initialization mode.");
	}

}

CSignalProcessingInstance * CSignalHandler::checkSignal (const std::string & sName)
{
		if (m_bIsInitializing)
			throw CException (eErrorCode::COULDNOTCHECKSIGNAL, "can not check signal, if in initialization mode.");

		auto iIter = m_SignalDefinitions.find (sName);
		if (iIter != m_SignalDefinitions.end ()) {
			auto pSignalDefinition = iIter->second;

			return pSignalDefinition->checkSignal ();
		}

		throw CException (eErrorCode::SIGNALDEFINITIONNOTFOUND, "signal definition not found: " + sName);

	}

CSignalSendInstance * CSignalHandler::prepareSignal (const std::string & sName)
{
	if (m_bIsInitializing)
		throw CException (eErrorCode::COULDNOTPREPARESIGNAL, "can not prepare signal, if in initialization mode.");

	auto iIter = m_SignalDefinitions.find (sName);
	if (iIter != m_SignalDefinitions.end ()) {
		auto pSignalDefinition = iIter->second;

		return pSignalDefinition->prepareSignal ();
	}

	throw CException (eErrorCode::SIGNALDEFINITIONNOTFOUND, "signal definition not found: " + sName);

}

void CSignalHandler::buildInstances ()
{
	if (m_bIsInitializing) {

		for (auto iIter : m_SignalDefinitions)
			iIter.second->buildInstances ();

		m_bIsInitializing = false;

	} else {
		throw CException (eErrorCode::CANNOTBUILDSIGNALINSTANCES, "signal instances have already been built.");
	}
}

void CSignalHandler::releaseExpiredSignals ()
{
	for (auto iIter : m_SignalDefinitions)
		iIter.second->releaseExpiredSignals ();
}

}
```
